	{attribute 'TcIecLibraryType'}
	{attribute 'external_name' := 'F_VN_GetAt_TcVnVector4_DINT_GUID_761AB84D_C513_5B06_61E4_80F931BBB792'}
	(* Gets the TcVnVector4_DINT element at the specified index of the container. *)
	FUNCTION F_VN_GetAt_TcVnVector4_DINT : HRESULT
	VAR_INPUT
		ipContainer	:	ITcVnContainer;	(* Container with TcVnVector4_DINT elements *)
		aElement	:	REFERENCE TO TcVnVector4_DINT;	(* Returns the element at the specified index *)
		nIndex	:	ULINT;	(* Index of the requested element *)
		hrPrev	:	HRESULT;	(* HRESULT indicating the result of previous operations (If SUCCEEDED(hrPrev) equals false, no operation is executed.) *)
	END_VAR

END_FUNCTION

// Functions/Basic Container Operations/F_VN_GetAt/F_VN_GetAt_TcVnVector4_LREAL

	{attribute 'TcIecLibraryType'}
	{attribute 'external_name' := 'F_VN_GetAt_TcVnVector4_LREAL_GUID_5FDC4290_5703_5BA7_61DD_065C1D8ADDFE'}
	(* Gets the TcVnVector4_LREAL element at the specified index of the container. *)
	FUNCTION F_VN_GetAt_TcVnVector4_LREAL : HRESULT
	VAR_INPUT
		ipContainer	:	ITcVnContainer;	(* Container with TcVnVector4_LREAL elements *)
		aElement	:	REFERENCE TO TcVnVector4_LREAL;	(* Returns the element at the specified index *)
		nIndex	:	ULINT;	(* Index of the requested element *)
		hrPrev	:	HRESULT;	(* HRESULT indicating the result of previous operations (If SUCCEEDED(hrPrev) equals false, no operation is executed.) *)
	END_VAR

END_FUNCTION

// Functions/Basic Container Operations/F_VN_GetAt/F_VN_GetAt_UDINT

	{attribute 'TcIecLibraryType'}
	{attribute 'external_name' := 'F_VN_GetAt_UDINT_GUID_C440DBA3_7390_5B33_575A_EBCC8FB96E53'}
	(* Gets the UDINT element at the specified index of the container. *)
	FUNCTION F_VN_GetAt_UDINT : HRESULT
	VAR_INPUT
		ipContainer	:	ITcVnContainer;	(* Container with UDINT elements *)
		nElement	:	REFERENCE TO UDINT;	(* Returns the element at the specified index *)
		nIndex	:	ULINT;	(* Index of the requested element *)
		hrPrev	:	HRESULT;	(* HRESULT indicating the result of previous operations (If SUCCEEDED(hrPrev) equals false, no operation is executed.) *)
	END_VAR

END_FUNCTION

// Functions/Basic Container Operations/F_VN_GetAt/F_VN_GetAt_ULINT

	{attribute 'TcIecLibraryType'}
	{attribute 'external_name' := 'F_VN_GetAt_ULINT_GUID_C7670D70_FA4B_5664_569F_3BAC6764E342'}
	(* Gets the ULINT element at the specified index of the container. *)
	FUNCTION F_VN_GetAt_ULINT : HRESULT
	VAR_INPUT
		ipContainer	:	ITcVnContainer;	(* Container with ULINT elements *)
		nElement	:	REFERENCE TO ULINT;	(* Returns the element at the specified index *)
		nIndex	:	ULINT;	(* Index of the requested element *)
		hrPrev	:	HRESULT;	(* HRESULT indicating the result of previous operations (If SUCCEEDED(hrPrev) equals false, no operation is executed.) *)
	END_VAR

END_FUNCTION

// Functions/Basic Container Operations/F_VN_InsertIntoContainer/F_VN_InsertIntoContainer_ITcVnContainer

	{attribute 'TcIecLibraryType'}
	{attribute 'external_name' := 'F_VN_InsertIntoContainer_ITcVnContainer_GUID_DDDC9785_B003_5B61_64D8_7B702B9B58A1'}
	(* Insert an element (or a range of elements) into a container before the specified position. *)
	FUNCTION F_VN_InsertIntoContainer_ITcVnContainer : HRESULT
	VAR_INPUT
		ipElement	:	ITcVnContainer;	(* Single element to insert into ipContainer or container with several elements *)
		ipContainer	:	ITcVnContainer;	(* Container in which to insert the element *)
		nIndex	:	ULINT;	(* Position, before which the element will be inserted *)
		hrPrev	:	HRESULT;	(* HRESULT indicating the result of previous operations (If SUCCEEDED(hrPrev) equals false, no operation is executed.) *)
	END_VAR

END_FUNCTION

// Functions/Basic Container Operations/F_VN_InsertIntoContainer/F_VN_InsertIntoContainer_ITcVnForwardIterator

	{attribute 'TcIecLibraryType'}
	{attribute 'external_name' := 'F_VN_InsertIntoContainer_ITcVnForwardIterator_GUID_80A27022_E316_5DC3_60F7_8E6960A418A2'}
	(* Insert an element (represented by an iterator) into a container before the specified position. *)
	FUNCTION F_VN_InsertIntoContainer_ITcVnForwardIterator : HRESULT
	VAR_INPUT
		ipElement	:	ITcVnForwardIterator;	(* Single element to insert into ipContainer *)
		ipContainer	:	ITcVnContainer;	(* Container in which to insert the element *)
		nIndex	:	ULINT;	(* Position, before which the element will be inserted *)
		hrPrev	:	HRESULT;	(* HRESULT indicating the result of previous operations (If SUCCEEDED(hrPrev) equals false, no operation is executed.) *)
	END_VAR

END_FUNCTION

// Functions/Basic Container Operations/F_VN_InsertIntoContainer/F_VN_InsertIntoContainer_DINT

	{attribute 'TcIecLibraryType'}
	{attribute 'external_name' := 'F_VN_InsertIntoContainer_DINT_GUID_EFA0F64D_773F_5851_76D4_98F1756231A4'}
	(* Insert an element of type DINT into a container before the specified position. *)
	FUNCTION F_VN_InsertIntoContainer_DINT : HRESULT
	VAR_INPUT
		nElement	:	DINT;	(* Single element to insert into ipContainer *)
		ipContainer	:	ITcVnContainer;	(* Container in which to insert the element *)
		nIndex	:	ULINT;	(* Position, before which the element will be inserted *)
		hrPrev	:	HRESULT;	(* HRESULT indicating the result of previous operations (If SUCCEEDED(hrPrev) equals false, no operation is executed.) *)
	END_VAR

END_FUNCTION

// Functions/Basic Container Operations/F_VN_InsertIntoContainer/F_VN_InsertIntoContainer_LREAL

	{attribute 'TcIecLibraryType'}
	{attribute 'external_name' := 'F_VN_InsertIntoContainer_LREAL_GUID_72B81CEB_6BEB_5915_6CF4_FBE0016B575A'}
	(* Insert an element of type LREAL into a container before the specified position. *)
	FUNCTION F_VN_InsertIntoContainer_LREAL : HRESULT
	VAR_INPUT
		fElement	:	LREAL;	(* Single element to insert into ipContainer *)
		ipContainer	:	ITcVnContainer;	(* Container in which to insert the element *)
		nIndex	:	ULINT;	(* Position, before which the element will be inserted *)
		hrPrev	:	HRESULT;	(* HRESULT indicating the result of previous operations (If SUCCEEDED(hrPrev) equals false, no operation is executed.) *)
	END_VAR

END_FUNCTION

// Functions/Basic Container Operations/F_VN_InsertIntoContainer/F_VN_InsertIntoContainer_REAL

	{attribute 'TcIecLibraryType'}
	{attribute 'external_name' := 'F_VN_InsertIntoContainer_REAL_GUID_3EA6CA06_995B_58CA_78EF_95938B01338C'}
	(* Insert an element of type REAL into a container before the specified position. *)
	FUNCTION F_VN_InsertIntoContainer_REAL : HRESULT
	VAR_INPUT
		fElement	:	REAL;	(* Single element to insert into ipContainer *)
		ipContainer	:	ITcVnContainer;	(* Container in which to insert the element *)
		nIndex	:	ULINT;	(* Position, before which the element will be inserted *)
		hrPrev	:	HRESULT;	(* HRESULT indicating the result of previous operations (If SUCCEEDED(hrPrev) equals false, no operation is executed.) *)
	END_VAR

END_FUNCTION

// Functions/Basic Container Operations/F_VN_InsertIntoContainer/F_VN_InsertIntoContainer_SINT

	{attribute 'TcIecLibraryType'}
	{attribute 'external_name' := 'F_VN_InsertIntoContainer_SINT_GUID_DC281E74_0A3E_5FA1_760C_538B9F283AFE'}
	(* Insert an element of type SINT into a container before the specified position. *)
	FUNCTION F_VN_InsertIntoContainer_SINT : HRESULT
	VAR_INPUT
		nElement	:	SINT;	(* Single element to insert into ipContainer *)
		ipContainer	:	ITcVnContainer;	(* Container in which to insert the element *)
		nIndex	:	ULINT;	(* Position, before which the element will be inserted *)
		hrPrev	:	HRESULT;	(* HRESULT indicating the result of previous operations (If SUCCEEDED(hrPrev) equals false, no operation is executed.) *)
	END_VAR

END_FUNCTION

// Functions/Basic Container Operations/F_VN_InsertIntoContainer/F_VN_InsertIntoContainer_TcVnDMatch

	{attribute 'TcIecLibraryType'}
	{attribute 'external_name' := 'F_VN_InsertIntoContainer_TcVnDMatch_GUID_6288EBFB_184C_50FA_5092_D3D94B3EFDC4'}
	(* Insert an element of type TcVnDMatch into a container before the specified position. *)
	FUNCTION F_VN_InsertIntoContainer_TcVnDMatch : HRESULT
	VAR_INPUT
		stElement	:	REFERENCE TO TcVnDMatch;	(* Single element to insert into ipContainer *)
		ipContainer	:	ITcVnContainer;	(* Container in which to insert the element *)
		nIndex	:	ULINT;	(* Position, before which the element will be inserted *)
		hrPrev	:	HRESULT;	(* HRESULT indicating the result of previous operations (If SUCCEEDED(hrPrev) equals false, no operation is executed.) *)
	END_VAR

END_FUNCTION

// Functions/Basic Container Operations/F_VN_InsertIntoContainer/F_VN_InsertIntoContainer_TcVnKeyPoint

	{attribute 'TcIecLibraryType'}
	{attribute 'external_name' := 'F_VN_InsertIntoContainer_TcVnKeyPoint_GUID_B6243C78_DA27_5D5E_5D78_25085B9D62AA'}
	(* Insert an element of type TcVnKeyPoint into a container before the specified position. *)
	FUNCTION F_VN_InsertIntoContainer_TcVnKeyPoint : HRESULT
	VAR_INPUT
		stElement	:	REFERENCE TO TcVnKeyPoint;	(* Single element to insert into ipContainer *)
		ipContainer	:	ITcVnContainer;	(* Container in which to insert the element *)
		nIndex	:	ULINT;	(* Position, before which the element will be inserted *)
		hrPrev	:	HRESULT;	(* HRESULT indicating the result of previous operations (If SUCCEEDED(hrPrev) equals false, no operation is executed.) *)
	END_VAR

END_FUNCTION

// Functions/Basic Container Operations/F_VN_InsertIntoContainer/F_VN_InsertIntoContainer_TcVnPoint2_DINT

	{attribute 'TcIecLibraryType'}
	{attribute 'external_name' := 'F_VN_InsertIntoContainer_TcVnPoint2_DINT_GUID_F549CEB7_E5A4_5BCF_494B_F1B410216754'}
	(* Insert an element of type TcVnPoint2_DINT into a container before the specified position. *)
	FUNCTION F_VN_InsertIntoContainer_TcVnPoint2_DINT : HRESULT
	VAR_INPUT
		aElement	:	REFERENCE TO TcVnPoint2_DINT;	(* Single element to insert into ipContainer *)
		ipContainer	:	ITcVnContainer;	(* Container in which to insert the element *)
		nIndex	:	ULINT;	(* Position, before which the element will be inserted *)
		hrPrev	:	HRESULT;	(* HRESULT indicating the result of previous operations (If SUCCEEDED(hrPrev) equals false, no operation is executed.) *)
	END_VAR

END_FUNCTION

// Functions/Basic Container Operations/F_VN_InsertIntoContainer/F_VN_InsertIntoContainer_TcVnPoint2_LREAL

	{attribute 'TcIecLibraryType'}
	{attribute 'external_name' := 'F_VN_InsertIntoContainer_TcVnPoint2_LREAL_GUID_0F32A540_CDF3_51E7_5F9A_C73CAA45BBE6'}
	(* Insert an element of type TcVnPoint2_LREAL into a container before the specified position. *)
	FUNCTION F_VN_InsertIntoContainer_TcVnPoint2_LREAL : HRESULT
	VAR_INPUT
		aElement	:	REFERENCE TO TcVnPoint2_LREAL;	(* Single element to insert into ipContainer *)
		ipContainer	:	ITcVnContainer;	(* Container in which to insert the element *)
		nIndex	:	ULINT;	(* Position, before which the element will be inserted *)
		hrPrev	:	HRESULT;	(* HRESULT indicating the result of previous operations (If SUCCEEDED(hrPrev) equals false, no operation is executed.) *)
	END_VAR

END_FUNCTION

// Functions/Basic Container Operations/F_VN_InsertIntoContainer/F_VN_InsertIntoContainer_TcVnPoint2_REAL

	{attribute 'TcIecLibraryType'}
	{attribute 'external_name' := 'F_VN_InsertIntoContainer_TcVnPoint2_REAL_GUID_727FB356_9228_5964_747E_75B2553FC054'}
	(* Insert an element of type TcVnPoint2_REAL into a container before the specified position. *)
	FUNCTION F_VN_InsertIntoContainer_TcVnPoint2_REAL : HRESULT
	VAR_INPUT
		aElement	:	REFERENCE TO TcVnPoint2_REAL;	(* Single element to insert into ipContainer *)
		ipContainer	:	ITcVnContainer;	(* Container in which to insert the element *)
		nIndex	:	ULINT;	(* Position, before which the element will be inserted *)
		hrPrev	:	HRESULT;	(* HRESULT indicating the result of previous operations (If SUCCEEDED(hrPrev) equals false, no operation is executed.) *)
	END_VAR

END_FUNCTION

// Functions/Basic Container Operations/F_VN_InsertIntoContainer/F_VN_InsertIntoContainer_TcVnPoint3_LREAL

	{attribute 'TcIecLibraryType'}
	{attribute 'external_name' := 'F_VN_InsertIntoContainer_TcVnPoint3_LREAL_GUID_0773769E_E9AF_5176_7931_BF10F0216404'}
	(* Insert an element of type TcVnPoint3_LREAL into a container before the specified position. *)
	FUNCTION F_VN_InsertIntoContainer_TcVnPoint3_LREAL : HRESULT
	VAR_INPUT
		aElement	:	REFERENCE TO TcVnPoint3_LREAL;	(* Single element to insert into ipContainer *)
		ipContainer	:	ITcVnContainer;	(* Container in which to insert the element *)
		nIndex	:	ULINT;	(* Position, before which the element will be inserted *)
		hrPrev	:	HRESULT;	(* HRESULT indicating the result of previous operations (If SUCCEEDED(hrPrev) equals false, no operation is executed.) *)
	END_VAR

END_FUNCTION

// Functions/Basic Container Operations/F_VN_InsertIntoContainer/F_VN_InsertIntoContainer_TcVnPoint3_REAL

	{attribute 'TcIecLibraryType'}
	{attribute 'external_name' := 'F_VN_InsertIntoContainer_TcVnPoint3_REAL_GUID_66633B0B_D08D_5FFD_5D37_7264CA3DA6E2'}
	(* Insert an element of type TcVnPoint3_REAL into a container before the specified position. *)
	FUNCTION F_VN_InsertIntoContainer_TcVnPoint3_REAL : HRESULT
	VAR_INPUT
		aElement	:	REFERENCE TO TcVnPoint3_REAL;	(* Single element to insert into ipContainer *)
		ipContainer	:	ITcVnContainer;	(* Container in which to insert the element *)
		nIndex	:	ULINT;	(* Position, before which the element will be inserted *)
		hrPrev	:	HRESULT;	(* HRESULT indicating the result of previous operations (If SUCCEEDED(hrPrev) equals false, no operation is executed.) *)
	END_VAR

END_FUNCTION

// Functions/Basic Container Operations/F_VN_InsertIntoContainer/F_VN_InsertIntoContainer_TcVnRectangle_DINT

	{attribute 'TcIecLibraryType'}
	{attribute 'external_name' := 'F_VN_InsertIntoContainer_TcVnRectangle_DINT_GUID_6D3C63D8_23BD_51A3_6598_36E39846907A'}
	(* Insert an element of type TcVnRectangle_DINT into a container before the specified position. *)
	FUNCTION F_VN_InsertIntoContainer_TcVnRectangle_DINT : HRESULT
	VAR_INPUT
		stElement	:	REFERENCE TO TcVnRectangle_DINT;	(* Single element to insert into ipContainer *)
		ipContainer	:	ITcVnContainer;	(* Container in which to insert the element *)
		nIndex	:	ULINT;	(* Position, before which the element will be inserted *)
		hrPrev	:	HRESULT;	(* HRESULT indicating the result of previous operations (If SUCCEEDED(hrPrev) equals false, no operation is executed.) *)
	END_VAR

END_FUNCTION

// Functions/Basic Container Operations/F_VN_InsertIntoContainer/F_VN_InsertIntoContainer_TcVnVector2_DINT

	{attribute 'TcIecLibraryType'}
	{attribute 'external_name' := 'F_VN_InsertIntoContainer_TcVnVector2_DINT_GUID_96D338D9_676E_50ED_60DB_FA4FFC7FDF34'}
	(* Insert an element of type TcVnVector2_DINT into a container before the specified position. *)
	FUNCTION F_VN_InsertIntoContainer_TcVnVector2_DINT : HRESULT
	VAR_INPUT
		aElement	:	REFERENCE TO TcVnVector2_DINT;	(* Single element to insert into ipContainer *)
		ipContainer	:	ITcVnContainer;	(* Container in which to insert the element *)
		nIndex	:	ULINT;	(* Position, before which the element will be inserted *)
		hrPrev	:	HRESULT;	(* HRESULT indicating the result of previous operations (If SUCCEEDED(hrPrev) equals false, no operation is executed.) *)
	END_VAR

END_FUNCTION

// Functions/Basic Container Operations/F_VN_InsertIntoContainer/F_VN_InsertIntoContainer_TcVnVector2_REAL

	{attribute 'TcIecLibraryType'}
	{attribute 'external_name' := 'F_VN_InsertIntoContainer_TcVnVector2_REAL_GUID_E74110AF_F945_5767_778B_24D2186D1C41'}
	(* Insert an element of type TcVnVector2_REAL into a container before the specified position. *)
	FUNCTION F_VN_InsertIntoContainer_TcVnVector2_REAL : HRESULT
	VAR_INPUT
		aElement	:	REFERENCE TO TcVnVector2_REAL;	(* Single element to insert into ipContainer *)
		ipContainer	:	ITcVnContainer;	(* Container in which to insert the element *)
		nIndex	:	ULINT;	(* Position, before which the element will be inserted *)
		hrPrev	:	HRESULT;	(* HRESULT indicating the result of previous operations (If SUCCEEDED(hrPrev) equals false, no operation is executed.) *)
	END_VAR

END_FUNCTION

// Functions/Basic Container Operations/F_VN_InsertIntoContainer/F_VN_InsertIntoContainer_TcVnVector3_REAL

	{attribute 'TcIecLibraryType'}
	{attribute 'external_name' := 'F_VN_InsertIntoContainer_TcVnVector3_REAL_GUID_7E113FC2_5BBC_54D7_6CFE_D698D46CE2A1'}
	(* Insert an element of type TcVnVector3_REAL into a container before the specified position. *)
	FUNCTION F_VN_InsertIntoContainer_TcVnVector3_REAL : HRESULT
	VAR_INPUT
		aElement	:	REFERENCE TO TcVnVector3_REAL;	(* Single element to insert into ipContainer *)
		ipContainer	:	ITcVnContainer;	(* Container in which to insert the element *)
		nIndex	:	ULINT;	(* Position, before which the element will be inserted *)
		hrPrev	:	HRESULT;	(* HRESULT indicating the result of previous operations (If SUCCEEDED(hrPrev) equals false, no operation is executed.) *)
	END_VAR

END_FUNCTION

// Functions/Basic Container Operations/F_VN_InsertIntoContainer/F_VN_InsertIntoContainer_TcVnVector4_DINT

	{attribute 'TcIecLibraryType'}
	{attribute 'external_name' := 'F_VN_InsertIntoContainer_TcVnVector4_DINT_GUID_4A3AD761_60B4_5081_5C01_BA7FAA99BCB9'}
	(* Insert an element of type TcVnVector4_DINT into a container before the specified position. *)
	FUNCTION F_VN_InsertIntoContainer_TcVnVector4_DINT : HRESULT
	VAR_INPUT
		aElement	:	REFERENCE TO TcVnVector4_DINT;	(* Single element to insert into ipContainer *)
		ipContainer	:	ITcVnContainer;	(* Container in which to insert the element *)
		nIndex	:	ULINT;	(* Position, before which the element will be inserted *)
		hrPrev	:	HRESULT;	(* HRESULT indicating the result of previous operations (If SUCCEEDED(hrPrev) equals false, no operation is executed.) *)
	END_VAR

END_FUNCTION

// Functions/Basic Container Operations/F_VN_InsertIntoContainer/F_VN_InsertIntoContainer_TcVnVector4_LREAL

	{attribute 'TcIecLibraryType'}
	{attribute 'external_name' := 'F_VN_InsertIntoContainer_TcVnVector4_LREAL_GUID_0DE3BAA5_BCB8_5749_62E9_D0780F00C723'}
	(* Insert an element of type TcVnVector4_LREAL into a container before the specified position. *)
	FUNCTION F_VN_InsertIntoContainer_TcVnVector4_LREAL : HRESULT
	VAR_INPUT
		aElement	:	REFERENCE TO TcVnVector4_LREAL;	(* Single element to insert into ipContainer *)
		ipContainer	:	ITcVnContainer;	(* Container in which to insert the element *)
		nIndex	:	ULINT;	(* Position, before which the element will be inserted *)
		hrPrev	:	HRESULT;	(* HRESULT indicating the result of previous operations (If SUCCEEDED(hrPrev) equals false, no operation is executed.) *)
	END_VAR

END_FUNCTION

// Functions/Basic Container Operations/F_VN_InsertIntoContainer/F_VN_InsertIntoContainer_UDINT

	{attribute 'TcIecLibraryType'}
	{attribute 'external_name' := 'F_VN_InsertIntoContainer_UDINT_GUID_B6D1E6FC_98F6_5CDB_5CC3_8811ED90DFDF'}
	(* Insert an element of type UDINT into a container before the specified position. *)
	FUNCTION F_VN_InsertIntoContainer_UDINT : HRESULT
	VAR_INPUT
		nElement	:	UDINT;	(* Single element to insert into ipContainer *)
		ipContainer	:	ITcVnContainer;	(* Container in which to insert the element *)
		nIndex	:	ULINT;	(* Position, before which the element will be inserted *)
		hrPrev	:	HRESULT;	(* HRESULT indicating the result of previous operations (If SUCCEEDED(hrPrev) equals false, no operation is executed.) *)
	END_VAR

END_FUNCTION

// Functions/Basic Container Operations/F_VN_InsertIntoContainer/F_VN_InsertIntoContainer_ULINT

	{attribute 'TcIecLibraryType'}
	{attribute 'external_name' := 'F_VN_InsertIntoContainer_ULINT_GUID_0DA88F93_3472_5D7A_5EDC_DFF2F9A1782F'}
	(* Insert an element of type ULINT into a container before the specified position. *)
	FUNCTION F_VN_InsertIntoContainer_ULINT : HRESULT
	VAR_INPUT
		nElement	:	ULINT;	(* Single element to insert into ipContainer *)
		ipContainer	:	ITcVnContainer;	(* Container in which to insert the element *)
		nIndex	:	ULINT;	(* Position, before which the element will be inserted *)
		hrPrev	:	HRESULT;	(* HRESULT indicating the result of previous operations (If SUCCEEDED(hrPrev) equals false, no operation is executed.) *)
	END_VAR

END_FUNCTION

// Functions/Basic Container Operations/F_VN_SetAt/F_VN_SetAt_ITcVnContainer

	{attribute 'TcIecLibraryType'}
	{attribute 'external_name' := 'F_VN_SetAt_ITcVnContainer_GUID_476292B8_B77C_54F1_6FFA_C3AAC9D44D9F'}
	(* Sets the element at the specified index of the container. (Alternatively use interface method .SetAt.) *)
	FUNCTION F_VN_SetAt_ITcVnContainer : HRESULT
	VAR_INPUT
		ipElement	:	ITcVnContainer;	(* Element to set at the specified container position *)
		ipContainer	:	ITcVnContainer;	(* Container with ITcVnContainer elements, in which the element at position nIndex is replaced by ipElement *)
		nIndex	:	ULINT;	(* Index *)
		hrPrev	:	HRESULT;	(* HRESULT indicating the result of previous operations (If SUCCEEDED(hrPrev) equals false, no operation is executed.) *)
	END_VAR

END_FUNCTION

// Functions/Basic Container Operations/F_VN_SetAt/F_VN_SetAt_DINT

	{attribute 'TcIecLibraryType'}
	{attribute 'external_name' := 'F_VN_SetAt_DINT_GUID_D681C79A_99FB_542C_5064_21278FC65E88'}
	(* Sets the element at the specified index of the container. *)
	FUNCTION F_VN_SetAt_DINT : HRESULT
	VAR_INPUT
		nElement	:	DINT;	(* Element to set at the specified container position *)
		ipContainer	:	ITcVnContainer;	(* Container with DINT elements, in which the element at position nIndex is replaced by nElement *)
		nIndex	:	ULINT;	(* Index *)
		hrPrev	:	HRESULT;	(* HRESULT indicating the result of previous operations (If SUCCEEDED(hrPrev) equals false, no operation is executed.) *)
	END_VAR

END_FUNCTION

// Functions/Basic Container Operations/F_VN_SetAt/F_VN_SetAt_LREAL

	{attribute 'TcIecLibraryType'}
	{attribute 'external_name' := 'F_VN_SetAt_LREAL_GUID_423656CE_3EEB_50CE_538A_C2294F8AC9E8'}
	(* Sets the element at the specified index of the container. *)
	FUNCTION F_VN_SetAt_LREAL : HRESULT
	VAR_INPUT
		fElement	:	LREAL;	(* Element to set at the specified container position *)
		ipContainer	:	ITcVnContainer;	(* Container with LREAL elements, in which the element at position nIndex is replaced by fElement *)
		nIndex	:	ULINT;	(* Index *)
		hrPrev	:	HRESULT;	(* HRESULT indicating the result of previous operations (If SUCCEEDED(hrPrev) equals false, no operation is executed.) *)
	END_VAR

END_FUNCTION

// Functions/Basic Container Operations/F_VN_SetAt/F_VN_SetAt_REAL

	{attribute 'TcIecLibraryType'}
	{attribute 'external_name' := 'F_VN_SetAt_REAL_GUID_8D20883B_2232_5CA0_46F3_1CAEEB220474'}
	(* Sets the element at the specified index of the container. *)
	FUNCTION F_VN_SetAt_REAL : HRESULT
	VAR_INPUT
		fElement	:	REAL;	(* Element to set at the specified container position *)
		ipContainer	:	ITcVnContainer;	(* Container with REAL elements, in which the element at position nIndex is replaced by fElement *)
		nIndex	:	ULINT;	(* Index *)
		hrPrev	:	HRESULT;	(* HRESULT indicating the result of previous operations (If SUCCEEDED(hrPrev) equals false, no operation is executed.) *)
	END_VAR

END_FUNCTION

// Functions/Basic Container Operations/F_VN_SetAt/F_VN_SetAt_SINT

	{attribute 'TcIecLibraryType'}
	{attribute 'external_name' := 'F_VN_SetAt_SINT_GUID_53FC7629_B651_5D0C_6E10_8210E70EB0CE'}
	(* Sets the element at the specified index of the container. *)
	FUNCTION F_VN_SetAt_SINT : HRESULT
	VAR_INPUT
		nElement	:	SINT;	(* Element to set at the specified container position *)
		ipContainer	:	ITcVnContainer;	(* Container with SINT elements, in which the element at position nIndex is replaced by nElement *)
		nIndex	:	ULINT;	(* Index *)
		hrPrev	:	HRESULT;	(* HRESULT indicating the result of previous operations (If SUCCEEDED(hrPrev) equals false, no operation is executed.) *)
	END_VAR

END_FUNCTION

// Functions/Basic Container Operations/F_VN_SetAt/F_VN_SetAt_TcVnDMatch

	{attribute 'TcIecLibraryType'}
	{attribute 'external_name' := 'F_VN_SetAt_TcVnDMatch_GUID_DE6374D9_34B5_5A1A_76F3_D708397AF9E9'}
	(* Sets the element at the specified index of the container. *)
	FUNCTION F_VN_SetAt_TcVnDMatch : HRESULT
	VAR_INPUT
		stElement	:	REFERENCE TO TcVnDMatch;	(* Element to set at the specified container position *)
		ipContainer	:	ITcVnContainer;	(* Container with TcVnDMatch elements, in which the element at position nIndex is replaced by stElement *)
		nIndex	:	ULINT;	(* Index *)
		hrPrev	:	HRESULT;	(* HRESULT indicating the result of previous operations (If SUCCEEDED(hrPrev) equals false, no operation is executed.) *)
	END_VAR

END_FUNCTION

// Functions/Basic Container Operations/F_VN_SetAt/F_VN_SetAt_TcVnKeyPoint

	{attribute 'TcIecLibraryType'}
	{attribute 'external_name' := 'F_VN_SetAt_TcVnKeyPoint_GUID_A6F74671_C5E7_5652_6D51_85B28D5B5475'}
	(* Sets the element at the specified index of the container. *)
	FUNCTION F_VN_SetAt_TcVnKeyPoint : HRESULT
	VAR_INPUT
		stElement	:	REFERENCE TO TcVnKeyPoint;	(* Element to set at the specified container position *)
		ipContainer	:	ITcVnContainer;	(* Container with TcVnKeyPoint elements, in which the element at position nIndex is replaced by stElement *)
		nIndex	:	ULINT;	(* Index *)
		hrPrev	:	HRESULT;	(* HRESULT indicating the result of previous operations (If SUCCEEDED(hrPrev) equals false, no operation is executed.) *)
	END_VAR

END_FUNCTION

// Functions/Basic Container Operations/F_VN_SetAt/F_VN_SetAt_TcVnPoint2_DINT

	{attribute 'TcIecLibraryType'}
	{attribute 'external_name' := 'F_VN_SetAt_TcVnPoint2_DINT_GUID_CBB9CE79_18E6_5A86_53EC_DCC9DA313DFD'}
	(* Sets the element at the specified index of the container. *)
	FUNCTION F_VN_SetAt_TcVnPoint2_DINT : HRESULT
	VAR_INPUT
		aElement	:	REFERENCE TO TcVnPoint2_DINT;	(* Element to set at the specified container position *)
		ipContainer	:	ITcVnContainer;	(* Container with TcVnPoint2_DINT elements, in which the element at position nIndex is replaced by aElement *)
		nIndex	:	ULINT;	(* Index *)
		hrPrev	:	HRESULT;	(* HRESULT indicating the result of previous operations (If SUCCEEDED(hrPrev) equals false, no operation is executed.) *)
	END_VAR

END_FUNCTION

// Functions/Basic Container Operations/F_VN_SetAt/F_VN_SetAt_TcVnPoint2_LREAL

	{attribute 'TcIecLibraryType'}
	{attribute 'external_name' := 'F_VN_SetAt_TcVnPoint2_LREAL_GUID_C0803B4C_5E0A_59E7_4B96_60DFDE71D332'}
	(* Sets the element at the specified index of the container. *)
	FUNCTION F_VN_SetAt_TcVnPoint2_LREAL : HRESULT
	VAR_INPUT
		aElement	:	REFERENCE TO TcVnPoint2_LREAL;	(* Element to set at the specified container position *)
		ipContainer	:	ITcVnContainer;	(* Container with TcVnPoint2_LREAL elements, in which the element at position nIndex is replaced by aElement *)
		nIndex	:	ULINT;	(* Index *)
		hrPrev	:	HRESULT;	(* HRESULT indicating the result of previous operations (If SUCCEEDED(hrPrev) equals false, no operation is executed.) *)
	END_VAR

END_FUNCTION

// Functions/Basic Container Operations/F_VN_SetAt/F_VN_SetAt_TcVnPoint2_REAL

	{attribute 'TcIecLibraryType'}
	{attribute 'external_name' := 'F_VN_SetAt_TcVnPoint2_REAL_GUID_9089A3D2_ECED_55A2_704E_02C6F5AC1EC2'}
	(* Sets the element at the specified index of the container. *)
	FUNCTION F_VN_SetAt_TcVnPoint2_REAL : HRESULT
	VAR_INPUT
		aElement	:	REFERENCE TO TcVnPoint2_REAL;	(* Element to set at the specified container position *)
		ipContainer	:	ITcVnContainer;	(* Container with TcVnPoint2_REAL elements, in which the element at position nIndex is replaced by aElement *)
		nIndex	:	ULINT;	(* Index *)
		hrPrev	:	HRESULT;	(* HRESULT indicating the result of previous operations (If SUCCEEDED(hrPrev) equals false, no operation is executed.) *)
	END_VAR

END_FUNCTION

// Functions/Basic Container Operations/F_VN_SetAt/F_VN_SetAt_TcVnPoint3_LREAL

	{attribute 'TcIecLibraryType'}
	{attribute 'external_name' := 'F_VN_SetAt_TcVnPoint3_LREAL_GUID_09B386C3_A97A_58B8_78DB_33FA210F652E'}
	(* Sets the element at the specified index of the container. *)
	FUNCTION F_VN_SetAt_TcVnPoint3_LREAL : HRESULT
	VAR_INPUT
		aElement	:	REFERENCE TO TcVnPoint3_LREAL;	(* Element to set at the specified container position *)
		ipContainer	:	ITcVnContainer;	(* Container with TcVnPoint3_LREAL elements, in which the element at position nIndex is replaced by aElement *)
		nIndex	:	ULINT;	(* Index *)
		hrPrev	:	HRESULT;	(* HRESULT indicating the result of previous operations (If SUCCEEDED(hrPrev) equals false, no operation is executed.) *)
	END_VAR

END_FUNCTION

// Functions/Basic Container Operations/F_VN_SetAt/F_VN_SetAt_TcVnPoint3_REAL

	{attribute 'TcIecLibraryType'}
	{attribute 'external_name' := 'F_VN_SetAt_TcVnPoint3_REAL_GUID_3AA6ED5C_D431_57BB_42D3_FC455BD67AEE'}
	(* Sets the element at the specified index of the container. *)
	FUNCTION F_VN_SetAt_TcVnPoint3_REAL : HRESULT
	VAR_INPUT
		aElement	:	REFERENCE TO TcVnPoint3_REAL;	(* Element to set at the specified container position *)
		ipContainer	:	ITcVnContainer;	(* Container with TcVnPoint3_REAL elements, in which the element at position nIndex is replaced by aElement *)
		nIndex	:	ULINT;	(* Index *)
		hrPrev	:	HRESULT;	(* HRESULT indicating the result of previous operations (If SUCCEEDED(hrPrev) equals false, no operation is executed.) *)
	END_VAR

END_FUNCTION

// Functions/Basic Container Operations/F_VN_SetAt/F_VN_SetAt_TcVnRectangle_DINT

	{attribute 'TcIecLibraryType'}
	{attribute 'external_name' := 'F_VN_SetAt_TcVnRectangle_DINT_GUID_B6875C80_57A2_53FA_62B0_D1707619700F'}
	(* Sets the element at the specified index of the container. *)
	FUNCTION F_VN_SetAt_TcVnRectangle_DINT : HRESULT
	VAR_INPUT
		stElement	:	REFERENCE TO TcVnRectangle_DINT;	(* Element to set at the specified container position *)
		ipContainer	:	ITcVnContainer;	(* Container with TcVnRectangle_DINT elements, in which the element at position nIndex is replaced by stElement *)
		nIndex	:	ULINT;	(* Index *)
		hrPrev	:	HRESULT;	(* HRESULT indicating the result of previous operations (If SUCCEEDED(hrPrev) equals false, no operation is executed.) *)
	END_VAR

END_FUNCTION

// Functions/Basic Container Operations/F_VN_SetAt/F_VN_SetAt_TcVnVector2_DINT

	{attribute 'TcIecLibraryType'}
	{attribute 'external_name' := 'F_VN_SetAt_TcVnVector2_DINT_GUID_DD29B9CC_1FA7_59DE_5D6A_4BD213537E38'}
	(* Sets the element at the specified index of the container. *)
	FUNCTION F_VN_SetAt_TcVnVector2_DINT : HRESULT
	VAR_INPUT
		aElement	:	REFERENCE TO TcVnVector2_DINT;	(* Element to set at the specified container position *)
		ipContainer	:	ITcVnContainer;	(* Container with TcVnVector2_DINT elements, in which the element at position nIndex is replaced by aElement *)
		nIndex	:	ULINT;	(* Index *)
		hrPrev	:	HRESULT;	(* HRESULT indicating the result of previous operations (If SUCCEEDED(hrPrev) equals false, no operation is executed.) *)
	END_VAR

END_FUNCTION

// Functions/Basic Container Operations/F_VN_SetAt/F_VN_SetAt_TcVnVector2_REAL

	{attribute 'TcIecLibraryType'}
	{attribute 'external_name' := 'F_VN_SetAt_TcVnVector2_REAL_GUID_0F5B0DA0_1480_5F68_5940_945F4CF7A15F'}
	(* Sets the element at the specified index of the container. *)
	FUNCTION F_VN_SetAt_TcVnVector2_REAL : HRESULT
	VAR_INPUT
		aElement	:	REFERENCE TO TcVnVector2_REAL;	(* Element to set at the specified container position *)
		ipContainer	:	ITcVnContainer;	(* Container with TcVnVector2_REAL elements, in which the element at position nIndex is replaced by aElement *)
		nIndex	:	ULINT;	(* Index *)
		hrPrev	:	HRESULT;	(* HRESULT indicating the result of previous operations (If SUCCEEDED(hrPrev) equals false, no operation is executed.) *)
	END_VAR

END_FUNCTION

// Functions/Basic Container Operations/F_VN_SetAt/F_VN_SetAt_TcVnVector3_REAL

	{attribute 'TcIecLibraryType'}
	{attribute 'external_name' := 'F_VN_SetAt_TcVnVector3_REAL_GUID_1454F9B4_0602_5B69_5941_414084146024'}
	(* Sets the element at the specified index of the container. *)
	FUNCTION F_VN_SetAt_TcVnVector3_REAL : HRESULT
	VAR_INPUT
		aElement	:	REFERENCE TO TcVnVector3_REAL;	(* Element to set at the specified container position *)
		ipContainer	:	ITcVnContainer;	(* Container with TcVnVector3_REAL elements, in which the element at position nIndex is replaced by aElement *)
		nIndex	:	ULINT;	(* Index *)
		hrPrev	:	HRESULT;	(* HRESULT indicating the result of previous operations (If SUCCEEDED(hrPrev) equals false, no operation is executed.) *)
	END_VAR

END_FUNCTION

// Functions/Basic Container Operations/F_VN_SetAt/F_VN_SetAt_TcVnVector4_DINT

	{attribute 'TcIecLibraryType'}
	{attribute 'external_name' := 'F_VN_SetAt_TcVnVector4_DINT_GUID_072C4DDC_9BFD_5FA3_4604_24EC0CFA6015'}
	(* Sets the element at the specified index of the container. *)
	FUNCTION F_VN_SetAt_TcVnVector4_DINT : HRESULT
	VAR_INPUT
		aElement	:	REFERENCE TO TcVnVector4_DINT;	(* Element to set at the specified container position *)
		ipContainer	:	ITcVnContainer;	(* Container with TcVnVector4_DINT elements, in which the element at position nIndex is replaced by aElement *)
		nIndex	:	ULINT;	(* Index *)
		hrPrev	:	HRESULT;	(* HRESULT indicating the result of previous operations (If SUCCEEDED(hrPrev) equals false, no operation is executed.) *)
	END_VAR

END_FUNCTION

// Functions/Basic Container Operations/F_VN_SetAt/F_VN_SetAt_TcVnVector4_LREAL

	{attribute 'TcIecLibraryType'}
	{attribute 'external_name' := 'F_VN_SetAt_TcVnVector4_LREAL_GUID_30AA56D9_7C3C_5666_4E1F_B45235D14E59'}
	(* Sets the element at the specified index of the container. *)
	FUNCTION F_VN_SetAt_TcVnVector4_LREAL : HRESULT
	VAR_INPUT
		aElement	:	REFERENCE TO TcVnVector4_LREAL;	(* Element to set at the specified container position *)
		ipContainer	:	ITcVnContainer;	(* Container with TcVnVector4_LREAL elements, in which the element at position nIndex is replaced by aElement *)
		nIndex	:	ULINT;	(* Index *)
		hrPrev	:	HRESULT;	(* HRESULT indicating the result of previous operations (If SUCCEEDED(hrPrev) equals false, no operation is executed.) *)
	END_VAR

END_FUNCTION

// Functions/Basic Container Operations/F_VN_SetAt/F_VN_SetAt_UDINT

	{attribute 'TcIecLibraryType'}
	{attribute 'external_name' := 'F_VN_SetAt_UDINT_GUID_40B05280_973C_5DCE_4051_62D4C4E38F07'}
	(* Sets the element at the specified index of the container. *)
	FUNCTION F_VN_SetAt_UDINT : HRESULT
	VAR_INPUT
		nElement	:	UDINT;	(* Element to set at the specified container position *)
		ipContainer	:	ITcVnContainer;	(* Container with UDINT elements, in which the element at position nIndex is replaced by nElement *)
		nIndex	:	ULINT;	(* Index *)
		hrPrev	:	HRESULT;	(* HRESULT indicating the result of previous operations (If SUCCEEDED(hrPrev) equals false, no operation is executed.) *)
	END_VAR

END_FUNCTION

// Functions/Basic Container Operations/F_VN_SetAt/F_VN_SetAt_ULINT

	{attribute 'TcIecLibraryType'}
	{attribute 'external_name' := 'F_VN_SetAt_ULINT_GUID_7FA306F3_87E6_5EB8_7DF2_7DE9EA11E389'}
	(* Sets the element at the specified index of the container. *)
	FUNCTION F_VN_SetAt_ULINT : HRESULT
	VAR_INPUT
		nElement	:	ULINT;	(* Element to set at the specified container position *)
		ipContainer	:	ITcVnContainer;	(* Container with ULINT elements, in which the element at position nIndex is replaced by nElement *)
		nIndex	:	ULINT;	(* Index *)
		hrPrev	:	HRESULT;	(* HRESULT indicating the result of previous operations (If SUCCEEDED(hrPrev) equals false, no operation is executed.) *)
	END_VAR

END_FUNCTION

// Functions/Geometric and Coordinate Transformations/Calibration/F_VN_CalibrateCamera

	{attribute 'TcIecLibraryType'}
	{attribute 'external_name' := 'F_VN_CalibrateCamera_GUID_689A4FD0_3F8C_52A9_6DE2_058A6325749E'}
	(* Compute the camera parameters (intrinsic + extrinsic) by evaluating an image containing a calibration pattern (circles). *)
	FUNCTION F_VN_CalibrateCamera : HRESULT
	VAR_INPUT
		ipSrcImage	:	ITcVnImage;	(* Source image containing a calibration pattern (1 channel, USINT elements) *)
		ipReferencePoints	:	ITcVnContainer;	(* Reference calibration pattern point positions (ContainerType_Vector_TcVnPoint3_REAL) *)
		aCameraMatrix	:	REFERENCE TO TcVnMatrix3x3_LREAL;	(* Returns the camera matrix *)
		aDistortionCoefficients	:	REFERENCE TO TcVnArray8_LREAL;	(* Returns the lens distortion coefficients [k1, k2, p1, p2, k3, k4, k5, k6] *)
		aRotationMatrix	:	REFERENCE TO TcVnMatrix3x3_LREAL;	(* Returns the rotation matrix *)
		aTranslationVector	:	REFERENCE TO TcVnVector3_LREAL;	(* Returns the translation vector *)
		fReprojError	:	REFERENCE TO LREAL;	(* Returns the reprojection error *)
		stBlobDetectionParams	:	REFERENCE TO TcVnParamsBlobDetection;	(* Parameters for the internally used F_VN_DetectBlobs function *)
		stCalibrationOptions	:	REFERENCE TO TcVnCameraCalibrationOptions;	(* Calibration options *)
		hrPrev	:	HRESULT;	(* HRESULT indicating the result of previous operations (If SUCCEEDED(hrPrev) equals false, no operation is executed.) *)
	END_VAR

END_FUNCTION

// Functions/Geometric and Coordinate Transformations/Calibration/F_VN_CalibrateCameraExp

	{attribute 'TcIecLibraryType'}
	{attribute 'external_name' := 'F_VN_CalibrateCameraExp_GUID_9E4F8F39_C817_5DF3_763A_2115BCB02FB8'}
	(* Compute the camera parameters (intrinsic + extrinsic) by evaluating images containing a calibration pattern (circles). The extrinsic parameters are computed for the first image in the array. (expert function) *)
	FUNCTION F_VN_CalibrateCameraExp : HRESULT
	VAR_INPUT
		pSrcImages	:	PVOID;	(* Pointer to an array of source images, each containing the same calibration pattern (1 channel, USINT elements) *)
		nSrcArraySize	:	UINT;	(* pSrcImages array size *)
		ipReferencePoints	:	ITcVnContainer;	(* Reference calibration pattern point positions (ContainerType_Vector_TcVnPoint3_REAL) *)
		aCameraMatrix	:	REFERENCE TO TcVnMatrix3x3_LREAL;	(* Returns the camera matrix *)
		aDistortionCoefficients	:	REFERENCE TO TcVnArray8_LREAL;	(* Returns the lens distortion coefficients [k1, k2, p1, p2, k3, k4, k5, k6] *)
		aRotationMatrix	:	REFERENCE TO TcVnMatrix3x3_LREAL;	(* Returns the rotation matrix *)
		aTranslationVector	:	REFERENCE TO TcVnVector3_LREAL;	(* Returns the translation vector *)
		fReprojError	:	REFERENCE TO LREAL;	(* Returns the reprojection error *)
		stBlobDetectionParams	:	REFERENCE TO TcVnParamsBlobDetection;	(* Parameters for the internally used F_VN_DetectBlobs function *)
		stCalibrationOptions	:	REFERENCE TO TcVnCameraCalibrationOptions;	(* Calibration options *)
		hrPrev	:	HRESULT;	(* HRESULT indicating the result of previous operations (If SUCCEEDED(hrPrev) equals false, no operation is executed.) *)
	END_VAR

END_FUNCTION

// Functions/Geometric and Coordinate Transformations/Calibration/F_VN_CalibrateCameraManually

	{attribute 'TcIecLibraryType'}
	{attribute 'external_name' := 'F_VN_CalibrateCameraManually_GUID_DE881DBF_7F98_560E_6A5A_763C7B294004'}
	(* Compute the camera parameters (intrinsic + extrinsic). *)
	FUNCTION F_VN_CalibrateCameraManually : HRESULT
	VAR_INPUT
		ipImagePoints	:	ITcVnContainer;	(* Provided image points of multiple images (ContainerType_Vector_Vector_TcVnPoint2_REAL, each inner container with at least 4 points, same order as in ipReferencePoints) *)
		nImageWidth	:	UDINT;	(* Image width *)
		nImageHeight	:	UDINT;	(* Image height *)
		ipReferencePoints	:	ITcVnContainer;	(* Reference world points (ContainerType_Vector_Vector_TcVnPoint3_REAL, same amount of points as ipImagePoints) *)
		aCameraMatrix	:	REFERENCE TO TcVnMatrix3x3_LREAL;	(* Returns the camera matrix *)
		aDistortionCoefficients	:	REFERENCE TO TcVnArray8_LREAL;	(* Returns the lens distortion coefficients [k1, k2, p1, p2, k3, k4, k5, k6] *)
		aRotationMatrix	:	REFERENCE TO TcVnMatrix3x3_LREAL;	(* Returns the rotation matrix *)
		aTranslationVector	:	REFERENCE TO TcVnVector3_LREAL;	(* Returns the translation vector *)
		fReprojError	:	REFERENCE TO LREAL;	(* Returns the reprojection error *)
		stCalibrationOptions	:	REFERENCE TO TcVnCameraCalibrationOptions;	(* Calibration options *)
		hrPrev	:	HRESULT;	(* HRESULT indicating the result of previous operations (If SUCCEEDED(hrPrev) equals false, no operation is executed.) *)
	END_VAR

END_FUNCTION

// Functions/Geometric and Coordinate Transformations/Calibration/F_VN_CalibrateCameraPlanar

	{attribute 'TcIecLibraryType'}
	{attribute 'external_name' := 'F_VN_CalibrateCameraPlanar_GUID_5EA61155_E866_5827_428A_3D35396EE97C'}
	(* Calibrate camera using a planar calibration pattern comprised of four circles marking the corners of a rectangle. *)
	FUNCTION F_VN_CalibrateCameraPlanar : HRESULT
	VAR_INPUT
		ipSrcImage	:	ITcVnImage;	(* Binary source image (background zero, markers non-zero) *)
		aMarkerPositions	:	REFERENCE TO TcVnArray4_Point2_REAL;	(* Marker positions within their plane using world units (right-handed coordinate system) *)
		aTransformationMatrix	:	REFERENCE TO TcVnMatrix3x3_LREAL;	(* Returns a 3-by-3 matrix for the transformation from image coordinates into the reference coordinate system *)
		hrPrev	:	HRESULT;	(* HRESULT indicating the result of previous operations (If SUCCEEDED(hrPrev) equals false, no operation is executed.) *)
	END_VAR

END_FUNCTION

// Functions/Geometric and Coordinate Transformations/Calibration/F_VN_CalibrateCameraPlanarExp

	{attribute 'TcIecLibraryType'}
	{attribute 'external_name' := 'F_VN_CalibrateCameraPlanarExp_GUID_FEC1C597_273C_5520_575C_D0D2115421C4'}
	(* Calibrate camera using a planar calibration pattern comprised of four circles marking the corners of a rectangle. (expert function) *)
	FUNCTION F_VN_CalibrateCameraPlanarExp : HRESULT
	VAR_INPUT
		ipSrcImage	:	ITcVnImage;	(* Binary source image (background zero, markers non-zero) *)
		aMarkerPositions	:	REFERENCE TO TcVnArray4_Point2_REAL;	(* Marker positions within their plane using world units (right-handed coordinate system) *)
		aTransformationMatrix	:	REFERENCE TO TcVnMatrix3x3_LREAL;	(* Returns a 3-by-3 matrix for the transformation from image coordinates into the reference coordinate system *)
		aMarkerImagePositions	:	REFERENCE TO TcVnArray4_Point2_REAL;	(* Returns the marker positions in image coordinates (left-handed coordinate system) *)
		nMinMarkerArea	:	UDINT;	(* Minimum area for the detection of markers (Smaller markers are ignored.) *)
		nMaxMarkerArea	:	UDINT;	(* Maximum area for the detection of markers (Larger markers are ignored.) *)
		fMaxMarkerEccentricity	:	LREAL;	(* Maximum eccenticity for the detection of markers (The eccentricity measures deviations from a round shape (eccentricity = 0: round object; eccentricity = 1.0:  linear object).) *)
		hrPrev	:	HRESULT;	(* HRESULT indicating the result of previous operations (If SUCCEEDED(hrPrev) equals false, no operation is executed.) *)
	END_VAR

END_FUNCTION

// Functions/Geometric and Coordinate Transformations/Calibration/F_VN_CompensateLensDistortion

	{attribute 'TcIecLibraryType'}
	{attribute 'external_name' := 'F_VN_CompensateLensDistortion_GUID_CBB1E0C9_72E1_5B3E_7EB2_FD89B201A4A5'}
	(* Transforms an image to compensate the lens distortion. *)
	FUNCTION F_VN_CompensateLensDistortion : HRESULT
	VAR_INPUT
		ipSrcImage	:	ITcVnImage;	(* Source image *)
		ipDestImage	:	REFERENCE TO ITcVnImage;	(* Destination image (An appropriate destination image will be created if required.) *)
		aCameraMatrix	:	REFERENCE TO TcVnMatrix3x3_LREAL;	(* Camera matrix containing the intrinsic parameters *)
		aDistortionCoefficients	:	REFERENCE TO TcVnArray4_LREAL;	(* Lens distortion coefficients [k1, k2, p1, p2] *)
		hrPrev	:	HRESULT;	(* HRESULT indicating the result of previous operations (If SUCCEEDED(hrPrev) equals false, no operation is executed.) *)
	END_VAR

END_FUNCTION

// Functions/Geometric and Coordinate Transformations/Calibration/F_VN_CompensateLensDistortionExp1

	{attribute 'TcIecLibraryType'}
	{attribute 'external_name' := 'F_VN_CompensateLensDistortionExp1_GUID_51CC86CE_2EC2_5725_7926_EA4CF3599825'}
	(* Transforms an image to compensate the lens distortion. (expert function) *)
	FUNCTION F_VN_CompensateLensDistortionExp1 : HRESULT
	VAR_INPUT
		ipSrcImage	:	ITcVnImage;	(* Source image *)
		ipDestImage	:	REFERENCE TO ITcVnImage;	(* Destination image (An appropriate destination image will be created if required.) *)
		aCameraMatrix	:	REFERENCE TO TcVnMatrix3x3_LREAL;	(* Camera matrix containing the intrinsic parameters *)
		aDistortionCoefficients	:	REFERENCE TO TcVnArray8_LREAL;	(* Lens distortion coefficients [k1, k2, p1, p2, k3, k4, k5, k6] *)
		hrPrev	:	HRESULT;	(* HRESULT indicating the result of previous operations (If SUCCEEDED(hrPrev) equals false, no operation is executed.) *)
	END_VAR

END_FUNCTION

// Functions/Geometric and Coordinate Transformations/Calibration/F_VN_CompensateLensDistortionExp2

	{attribute 'TcIecLibraryType'}
	{attribute 'external_name' := 'F_VN_CompensateLensDistortionExp2_GUID_AE57D942_6BC7_5727_5D22_454B8EF06455'}
	(* Transforms an image to compensate the lens distortion. (expert function) *)
	FUNCTION F_VN_CompensateLensDistortionExp2 : HRESULT
	VAR_INPUT
		ipSrcImage	:	ITcVnImage;	(* Source image *)
		ipDestImage	:	REFERENCE TO ITcVnImage;	(* Destination image (An appropriate destination image will be created if required.) *)
		aCameraMatrix	:	REFERENCE TO TcVnMatrix3x3_LREAL;	(* Camera matrix containing the intrinsic parameters *)
		aDistortionCoefficients	:	REFERENCE TO TcVnArray8_LREAL;	(* Lens distortion coefficients [k1, k2, p1, p2, k3, k4, k5, k6] *)
		aNewCameraMatrix	:	REFERENCE TO TcVnMatrix3x3_LREAL;	(* Allows additional scaling and shifting of the result image *)
		hrPrev	:	HRESULT;	(* HRESULT indicating the result of previous operations (If SUCCEEDED(hrPrev) equals false, no operation is executed.) *)
	END_VAR

END_FUNCTION

// Functions/Geometric and Coordinate Transformations/Calibration/F_VN_CompensateLensDistortionForPoints

	{attribute 'TcIecLibraryType'}
	{attribute 'external_name' := 'F_VN_CompensateLensDistortionForPoints_GUID_76295BA5_956B_5713_4503_6A5E53895B3F'}
	(* Transforms point coordinates to compensate the lens distortion. *)
	FUNCTION F_VN_CompensateLensDistortionForPoints : HRESULT
	VAR_INPUT
		ipSrcPoints	:	ITcVnContainer;	(* Container with source point coordinates (ContainerType_Vector_TcVnPoint2_REAL or ContainerType_Vector_TcVnPoint2_DINT) *)
		ipDestPoints	:	REFERENCE TO ITcVnContainer;	(* Returns a container with the transformed point coordinates (ContainerType_Vector_TcVnPoint2_REAL) *)
		aCameraMatrix	:	REFERENCE TO TcVnMatrix3x3_LREAL;	(* Camera matrix containing the intrinsic parameters *)
		aDistortionCoefficients	:	REFERENCE TO TcVnArray4_LREAL;	(* Lens distortion coefficients [k1, k2, p1, p2] *)
		hrPrev	:	HRESULT;	(* HRESULT indicating the result of previous operations (If SUCCEEDED(hrPrev) equals false, no operation is executed.) *)
	END_VAR

END_FUNCTION

// Functions/Geometric and Coordinate Transformations/Calibration/F_VN_CompensateLensDistortionForPointsExp1

	{attribute 'TcIecLibraryType'}
	{attribute 'external_name' := 'F_VN_CompensateLensDistortionForPointsExp1_GUID_17DC8C11_965C_573B_7421_45C78A98F0B1'}
	(* Transforms point coordinates to compensate the lens distortion. (expert function) *)
	FUNCTION F_VN_CompensateLensDistortionForPointsExp1 : HRESULT
	VAR_INPUT
		ipSrcPoints	:	ITcVnContainer;	(* Container with source point coordinates (ContainerType_Vector_TcVnPoint2_REAL or ContainerType_Vector_TcVnPoint2_DINT) *)
		ipDestPoints	:	REFERENCE TO ITcVnContainer;	(* Returns a container with the transformed point coordinates (ContainerType_Vector_TcVnPoint2_REAL) *)
		aCameraMatrix	:	REFERENCE TO TcVnMatrix3x3_LREAL;	(* Camera matrix containing the intrinsic parameters *)
		aDistortionCoefficients	:	REFERENCE TO TcVnArray8_LREAL;	(* Lens distortion coefficients [k1, k2, p1, p2, k3, k4, k5, k6] *)
		hrPrev	:	HRESULT;	(* HRESULT indicating the result of previous operations (If SUCCEEDED(hrPrev) equals false, no operation is executed.) *)
	END_VAR

END_FUNCTION

// Functions/Geometric and Coordinate Transformations/Calibration/F_VN_CompensateLensDistortionForPointsExp2

	{attribute 'TcIecLibraryType'}
	{attribute 'external_name' := 'F_VN_CompensateLensDistortionForPointsExp2_GUID_580DD8FE_232B_5D0F_56A5_CB616AB70164'}
	(* Transforms point coordinates to compensate the lens distortion. (expert function) *)
	FUNCTION F_VN_CompensateLensDistortionForPointsExp2 : HRESULT
	VAR_INPUT
		ipSrcPoints	:	ITcVnContainer;	(* Container with source point coordinates (ContainerType_Vector_TcVnPoint2_REAL or ContainerType_Vector_TcVnPoint2_DINT) *)
		ipDestPoints	:	REFERENCE TO ITcVnContainer;	(* Returns a container with the transformed point coordinates (ContainerType_Vector_TcVnPoint2_REAL) *)
		aCameraMatrix	:	REFERENCE TO TcVnMatrix3x3_LREAL;	(* Camera matrix containing the intrinsic parameters *)
		aDistortionCoefficients	:	REFERENCE TO TcVnArray8_LREAL;	(* Lens distortion coefficients [k1, k2, p1, p2, k3, k4, k5, k6] *)
		aNewCameraMatrix	:	REFERENCE TO TcVnMatrix3x3_LREAL;	(* Allows additional shifting of the result point coordinates *)
		hrPrev	:	HRESULT;	(* HRESULT indicating the result of previous operations (If SUCCEEDED(hrPrev) equals false, no operation is executed.) *)
	END_VAR

END_FUNCTION

// Functions/Geometric and Coordinate Transformations/Calibration/F_VN_TransformCoordinatesPlanar_Container

	{attribute 'TcIecLibraryType'}
	{attribute 'external_name' := 'F_VN_TransformCoordinatesPlanar_Container_GUID_0B0CC95B_F42B_5C42_6508_29E6B8063DF0'}
	(* Compute real-world coordinates for given image points or vice versa. *)
	FUNCTION F_VN_TransformCoordinatesPlanar_Container : HRESULT
	VAR_INPUT
		ipSrcPoints	:	ITcVnContainer;	(* Container with 2D source points (TcVnPoint2_DINT or TcVnPoint2_REAL or TcVnPoint2_LREAL) *)
		ipDestPoints	:	REFERENCE TO ITcVnContainer;	(* Returns the transformed 2D points (TcVnPoint2_LREAL) *)
		aTransformationMatrix	:	REFERENCE TO TcVnMatrix3x3_LREAL;	(* Transformation matrix obtained with VnCalibrateCameraPlanar() or its inverse matrix obtained with VnInvertMatrix3x3() *)
		hrPrev	:	HRESULT;	(* HRESULT indicating the result of previous operations (If SUCCEEDED(hrPrev) equals false, no operation is executed.) *)
	END_VAR

END_FUNCTION

// Functions/Geometric and Coordinate Transformations/Calibration/F_VN_TransformCoordinatesPlanar_Point

	{attribute 'TcIecLibraryType'}
	{attribute 'external_name' := 'F_VN_TransformCoordinatesPlanar_Point_GUID_FFF67447_DBD8_5FA8_6BD4_F8748C59BC0A'}
	(* Compute real-world coordinates for a given image point or vice versa. *)
	FUNCTION F_VN_TransformCoordinatesPlanar_Point : HRESULT
	VAR_INPUT
		aSrcPoint	:	REFERENCE TO TcVnPoint2_LREAL;	(* Point in the source coordinate system *)
		aDestPoint	:	REFERENCE TO TcVnPoint2_LREAL;	(* Returns point in the destination coordinate system *)
		aTransformationMatrix	:	REFERENCE TO TcVnMatrix3x3_LREAL;	(* Transformation matrix obtained with VnCalibrateCameraPlanar() or its inverse matrix obtained with VnInvertMatrix3x3() *)
		hrPrev	:	HRESULT;	(* HRESULT indicating the result of previous operations (If SUCCEEDED(hrPrev) equals false, no operation is executed.) *)
	END_VAR

END_FUNCTION

// Functions/Geometric and Coordinate Transformations/Calibration/F_VN_TransformCoordinatesImageToWorld_Container

	{attribute 'TcIecLibraryType'}
	{attribute 'external_name' := 'F_VN_TransformCoordinatesImageToWorld_Container_GUID_389B6CAE_805D_5DE7_5A22_E1B341FFCFBA'}
	(* Transform 2D image point coordinates to 3D world coordinates (using intrinsic + extrinsic calibration results). *)
	FUNCTION F_VN_TransformCoordinatesImageToWorld_Container : HRESULT
	VAR_INPUT
		ipSrcPoints2D	:	ITcVnContainer;	(* Container with 2D source points (TcVnPoint2_DINT or TcVnPoint2_REAL or TcVnPoint2_LREAL) *)
		ipDestPoints3D	:	REFERENCE TO ITcVnContainer;	(* Returns the transformed 3D points (TcVnPoint3_LREAL) *)
		aCameraMatrix	:	REFERENCE TO TcVnMatrix3x3_LREAL;	(* 3x3 camera matrix containing the intrinsic parameters *)
		aDistortionCoefficients	:	REFERENCE TO TcVnArray8_LREAL;	(* Lens distortion coefficients [k1, k2, p1, p2, k3, k4, k5, k6] *)
		aRotationMatrix	:	REFERENCE TO TcVnMatrix3x3_LREAL;	(* 3x3 rotation matrix *)
		aTranslationVector	:	REFERENCE TO TcVnVector3_LREAL;	(* Translation vector *)
		fZ	:	LREAL;	(* z coordinate (world coordinate system) of the transformed points (0 would be at (toplevel) calibration pattern) *)
		hrPrev	:	HRESULT;	(* HRESULT indicating the result of previous operations (If SUCCEEDED(hrPrev) equals false, no operation is executed.) *)
	END_VAR

END_FUNCTION

// Functions/Geometric and Coordinate Transformations/Calibration/F_VN_TransformCoordinatesImageToWorld_Point

	{attribute 'TcIecLibraryType'}
	{attribute 'external_name' := 'F_VN_TransformCoordinatesImageToWorld_Point_GUID_EFB98558_B4AE_5C23_6CCF_F027CE21A2E4'}
	(* Transform 2D image point coordinate to 3D world coordinate (using intrinsic + extrinsic calibration results). *)
	FUNCTION F_VN_TransformCoordinatesImageToWorld_Point : HRESULT
	VAR_INPUT
		aSrcPoint	:	REFERENCE TO TcVnPoint2_LREAL;	(* Point in the image coordinate system *)
		aDestPoint	:	REFERENCE TO TcVnPoint3_LREAL;	(* Returns the point in the world coordinate system *)
		aCameraMatrix	:	REFERENCE TO TcVnMatrix3x3_LREAL;	(* 3x3 camera matrix containing the intrinsic parameters *)
		aDistortionCoefficients	:	REFERENCE TO TcVnArray8_LREAL;	(* Lens distortion coefficients [k1, k2, p1, p2, k3, k4, k5, k6] *)
		aRotationMatrix	:	REFERENCE TO TcVnMatrix3x3_LREAL;	(* 3x3 rotation matrix *)
		aTranslationVector	:	REFERENCE TO TcVnVector3_LREAL;	(* Translation vector *)
		fZ	:	LREAL;	(* z coordinate (world coordinate system) of the transformed points (0 would be at (toplevel) calibration pattern) *)
		hrPrev	:	HRESULT;	(* HRESULT indicating the result of previous operations (If SUCCEEDED(hrPrev) equals false, no operation is executed.) *)
	END_VAR

END_FUNCTION

// Functions/Geometric and Coordinate Transformations/Calibration/F_VN_TransformCoordinatesWorldToImage_Container

	{attribute 'TcIecLibraryType'}
	{attribute 'external_name' := 'F_VN_TransformCoordinatesWorldToImage_Container_GUID_AA8D71AA_9B5D_526B_6C5E_5E8EFE8E239A'}
	(* Transform 3D world coordinates to 2D image coordinates (using intrinsic + extrinsic calibration results). *)
	FUNCTION F_VN_TransformCoordinatesWorldToImage_Container : HRESULT
	VAR_INPUT
		ipSrcPoints3D	:	ITcVnContainer;	(* Container with 3D source points (TcVnPoint3_LREAL) *)
		ipDestPoints2D	:	REFERENCE TO ITcVnContainer;	(* Returns the transformed 2D points (TcVnPoint2_REAL or TcVnPoint2_DINT, depending on bInteger) *)
		aCameraMatrix	:	REFERENCE TO TcVnMatrix3x3_LREAL;	(* 3x3 camera matrix containing the intrinsic parameters *)
		aDistortionCoefficients	:	REFERENCE TO TcVnArray8_LREAL;	(* Lens distortion coefficients [k1, k2, p1, p2, k3, k4, k5, k6] *)
		aRotationMatrix	:	REFERENCE TO TcVnMatrix3x3_LREAL;	(* 3x3 rotation matrix *)
		aTranslationVector	:	REFERENCE TO TcVnVector3_LREAL;	(* Translation vector *)
		bInteger	:	BOOL;	(* Selects whether the function returns a container of TcVnPoint2_DINT or TcVnPoint2_REAL *)
		hrPrev	:	HRESULT;	(* HRESULT indicating the result of previous operations (If SUCCEEDED(hrPrev) equals false, no operation is executed.) *)
	END_VAR

END_FUNCTION

// Functions/Geometric and Coordinate Transformations/Calibration/F_VN_TransformCoordinatesWorldToImage_Point

	{attribute 'TcIecLibraryType'}
	{attribute 'external_name' := 'F_VN_TransformCoordinatesWorldToImage_Point_GUID_EEBF188A_B8B9_5909_6E01_AFD0BEADA794'}
	(* Transform 3D world coordinates to 2D image coordinates (using intrinsic + extrinsic calibration results). *)
	FUNCTION F_VN_TransformCoordinatesWorldToImage_Point : HRESULT
	VAR_INPUT
		aSrcPoint	:	REFERENCE TO TcVnPoint3_LREAL;	(* 3D source point (world coordinate system) *)
		aDestPoint	:	REFERENCE TO TcVnPoint2_REAL;	(* Returns the transformed 2D point (image coordinate system) *)
		aCameraMatrix	:	REFERENCE TO TcVnMatrix3x3_LREAL;	(* 3x3 camera matrix containing the intrinsic parameters *)
		aDistortionCoefficients	:	REFERENCE TO TcVnArray8_LREAL;	(* Lens distortion coefficients [k1, k2, p1, p2, k3, k4, k5, k6] *)
		aRotationMatrix	:	REFERENCE TO TcVnMatrix3x3_LREAL;	(* 3x3 rotation matrix *)
		aTranslationVector	:	REFERENCE TO TcVnVector3_LREAL;	(* Translation vector *)
		hrPrev	:	HRESULT;	(* HRESULT indicating the result of previous operations (If SUCCEEDED(hrPrev) equals false, no operation is executed.) *)
	END_VAR

END_FUNCTION

// Functions/Container Statistics/F_VN_MaxElementElementwise/F_VN_MaxElementElementwise_DINT

	{attribute 'TcIecLibraryType'}
	{attribute 'external_name' := 'F_VN_MaxElementElementwise_DINT_GUID_C98AF7AB_56CC_57E6_5493_B27637C0D032'}
	(* Gets the element wise maximum container element. *)
	FUNCTION F_VN_MaxElementElementwise_DINT : HRESULT
	VAR_INPUT
		ipContainer	:	ITcVnContainer;	(* Source container *)
		nMax	:	REFERENCE TO DINT;	(* Returns the requested element *)
		hrPrev	:	HRESULT;	(* HRESULT indicating the result of previous operations (If SUCCEEDED(hrPrev) equals false, no operation is executed.) *)
	END_VAR

END_FUNCTION

// Functions/Container Statistics/F_VN_MaxElementElementwise/F_VN_MaxElementElementwise_LREAL

	{attribute 'TcIecLibraryType'}
	{attribute 'external_name' := 'F_VN_MaxElementElementwise_LREAL_GUID_2A3E8EC8_F128_588A_6EE5_33C1A06A009C'}
	(* Gets the element wise maximum container element. *)
	FUNCTION F_VN_MaxElementElementwise_LREAL : HRESULT
	VAR_INPUT
		ipContainer	:	ITcVnContainer;	(* Source container *)
		fMax	:	REFERENCE TO LREAL;	(* Returns the requested element *)
		hrPrev	:	HRESULT;	(* HRESULT indicating the result of previous operations (If SUCCEEDED(hrPrev) equals false, no operation is executed.) *)
	END_VAR

END_FUNCTION

// Functions/Container Statistics/F_VN_MaxElementElementwise/F_VN_MaxElementElementwise_REAL

	{attribute 'TcIecLibraryType'}
	{attribute 'external_name' := 'F_VN_MaxElementElementwise_REAL_GUID_41CF3A3D_6549_55A9_63E5_D8722147DA12'}
	(* Gets the element wise maximum container element. *)
	FUNCTION F_VN_MaxElementElementwise_REAL : HRESULT
	VAR_INPUT
		ipContainer	:	ITcVnContainer;	(* Source container *)
		fMax	:	REFERENCE TO REAL;	(* Returns the requested element *)
		hrPrev	:	HRESULT;	(* HRESULT indicating the result of previous operations (If SUCCEEDED(hrPrev) equals false, no operation is executed.) *)
	END_VAR

END_FUNCTION

// Functions/Container Statistics/F_VN_MaxElementElementwise/F_VN_MaxElementElementwise_SINT

	{attribute 'TcIecLibraryType'}
	{attribute 'external_name' := 'F_VN_MaxElementElementwise_SINT_GUID_BF5E1168_B97B_5AA5_44C6_95FEA6EAEBE8'}
	(* Gets the element wise maximum container element. *)
	FUNCTION F_VN_MaxElementElementwise_SINT : HRESULT
	VAR_INPUT
		ipContainer	:	ITcVnContainer;	(* Source container *)
		nMax	:	REFERENCE TO SINT;	(* Returns the requested element *)
		hrPrev	:	HRESULT;	(* HRESULT indicating the result of previous operations (If SUCCEEDED(hrPrev) equals false, no operation is executed.) *)
	END_VAR

END_FUNCTION

// Functions/Container Statistics/F_VN_MaxElementElementwise/F_VN_MaxElementElementwise_TcVnPoint2_DINT

	{attribute 'TcIecLibraryType'}
	{attribute 'external_name' := 'F_VN_MaxElementElementwise_TcVnPoint2_DINT_GUID_C3B9FD32_728B_56A7_76C0_7A5C6C81DD31'}
	(* Gets the element wise maximum container element. *)
	FUNCTION F_VN_MaxElementElementwise_TcVnPoint2_DINT : HRESULT
	VAR_INPUT
		ipContainer	:	ITcVnContainer;	(* Source container *)
		aMax	:	REFERENCE TO TcVnPoint2_DINT;	(* Returns the requested element *)
		hrPrev	:	HRESULT;	(* HRESULT indicating the result of previous operations (If SUCCEEDED(hrPrev) equals false, no operation is executed.) *)
	END_VAR

END_FUNCTION

// Functions/Container Statistics/F_VN_MaxElementElementwise/F_VN_MaxElementElementwise_TcVnPoint2_LREAL

	{attribute 'TcIecLibraryType'}
	{attribute 'external_name' := 'F_VN_MaxElementElementwise_TcVnPoint2_LREAL_GUID_CDD9B01E_3E48_5636_53B6_DCE8899F5881'}
	(* Gets the element wise maximum container element. *)
	FUNCTION F_VN_MaxElementElementwise_TcVnPoint2_LREAL : HRESULT
	VAR_INPUT
		ipContainer	:	ITcVnContainer;	(* Source container *)
		aMax	:	REFERENCE TO TcVnPoint2_LREAL;	(* Returns the requested element *)
		hrPrev	:	HRESULT;	(* HRESULT indicating the result of previous operations (If SUCCEEDED(hrPrev) equals false, no operation is executed.) *)
	END_VAR

END_FUNCTION

// Functions/Container Statistics/F_VN_MaxElementElementwise/F_VN_MaxElementElementwise_TcVnPoint2_REAL

	{attribute 'TcIecLibraryType'}
	{attribute 'external_name' := 'F_VN_MaxElementElementwise_TcVnPoint2_REAL_GUID_6620B218_E936_5552_713C_BF3A14021415'}
	(* Gets the element wise maximum container element. *)
	FUNCTION F_VN_MaxElementElementwise_TcVnPoint2_REAL : HRESULT
	VAR_INPUT
		ipContainer	:	ITcVnContainer;	(* Source container *)
		aMax	:	REFERENCE TO TcVnPoint2_REAL;	(* Returns the requested element *)
		hrPrev	:	HRESULT;	(* HRESULT indicating the result of previous operations (If SUCCEEDED(hrPrev) equals false, no operation is executed.) *)
	END_VAR

END_FUNCTION

// Functions/Container Statistics/F_VN_MaxElementElementwise/F_VN_MaxElementElementwise_TcVnPoint3_LREAL

	{attribute 'TcIecLibraryType'}
	{attribute 'external_name' := 'F_VN_MaxElementElementwise_TcVnPoint3_LREAL_GUID_6275D7C0_5FF9_5B4F_527C_4C477599B2B3'}
	(* Gets the element wise maximum container element. *)
	FUNCTION F_VN_MaxElementElementwise_TcVnPoint3_LREAL : HRESULT
	VAR_INPUT
		ipContainer	:	ITcVnContainer;	(* Source container *)
		aMax	:	REFERENCE TO TcVnPoint3_LREAL;	(* Returns the requested element *)
		hrPrev	:	HRESULT;	(* HRESULT indicating the result of previous operations (If SUCCEEDED(hrPrev) equals false, no operation is executed.) *)
	END_VAR

END_FUNCTION

// Functions/Container Statistics/F_VN_MaxElementElementwise/F_VN_MaxElementElementwise_TcVnPoint3_REAL

	{attribute 'TcIecLibraryType'}
	{attribute 'external_name' := 'F_VN_MaxElementElementwise_TcVnPoint3_REAL_GUID_95A8C032_C8FF_5AE3_5557_6C399C5D237E'}
	(* Gets the element wise maximum container element. *)
	FUNCTION F_VN_MaxElementElementwise_TcVnPoint3_REAL : HRESULT
	VAR_INPUT
		ipContainer	:	ITcVnContainer;	(* Source container *)
		aMax	:	REFERENCE TO TcVnPoint3_REAL;	(* Returns the requested element *)
		hrPrev	:	HRESULT;	(* HRESULT indicating the result of previous operations (If SUCCEEDED(hrPrev) equals false, no operation is executed.) *)
	END_VAR

END_FUNCTION

// Functions/Container Statistics/F_VN_MaxElementElementwise/F_VN_MaxElementElementwise_TcVnVector2_DINT

	{attribute 'TcIecLibraryType'}
	{attribute 'external_name' := 'F_VN_MaxElementElementwise_TcVnVector2_DINT_GUID_ABD64B03_A5A7_5CA8_45E0_955D0270CCFB'}
	(* Gets the element wise maximum container element. *)
	FUNCTION F_VN_MaxElementElementwise_TcVnVector2_DINT : HRESULT
	VAR_INPUT
		ipContainer	:	ITcVnContainer;	(* Source container *)
		aMax	:	REFERENCE TO TcVnVector2_DINT;	(* Returns the requested element *)
		hrPrev	:	HRESULT;	(* HRESULT indicating the result of previous operations (If SUCCEEDED(hrPrev) equals false, no operation is executed.) *)
	END_VAR

END_FUNCTION

// Functions/Container Statistics/F_VN_MaxElementElementwise/F_VN_MaxElementElementwise_TcVnVector2_REAL

	{attribute 'TcIecLibraryType'}
	{attribute 'external_name' := 'F_VN_MaxElementElementwise_TcVnVector2_REAL_GUID_C54A6415_4011_506E_4571_CC593C6D6900'}
	(* Gets the element wise maximum container element. *)
	FUNCTION F_VN_MaxElementElementwise_TcVnVector2_REAL : HRESULT
	VAR_INPUT
		ipContainer	:	ITcVnContainer;	(* Source container *)
		aMax	:	REFERENCE TO TcVnVector2_REAL;	(* Returns the requested element *)
		hrPrev	:	HRESULT;	(* HRESULT indicating the result of previous operations (If SUCCEEDED(hrPrev) equals false, no operation is executed.) *)
	END_VAR

END_FUNCTION

// Functions/Container Statistics/F_VN_MaxElementElementwise/F_VN_MaxElementElementwise_TcVnVector3_REAL

	{attribute 'TcIecLibraryType'}
	{attribute 'external_name' := 'F_VN_MaxElementElementwise_TcVnVector3_REAL_GUID_F202B0FF_602F_510A_769F_B41F07A62490'}
	(* Gets the element wise maximum container element. *)
	FUNCTION F_VN_MaxElementElementwise_TcVnVector3_REAL : HRESULT
	VAR_INPUT
		ipContainer	:	ITcVnContainer;	(* Source container *)
		aMax	:	REFERENCE TO TcVnVector3_REAL;	(* Returns the requested element *)
		hrPrev	:	HRESULT;	(* HRESULT indicating the result of previous operations (If SUCCEEDED(hrPrev) equals false, no operation is executed.) *)
	END_VAR

END_FUNCTION

// Functions/Container Statistics/F_VN_MaxElementElementwise/F_VN_MaxElementElementwise_TcVnVector4_DINT

	{attribute 'TcIecLibraryType'}
	{attribute 'external_name' := 'F_VN_MaxElementElementwise_TcVnVector4_DINT_GUID_3E877F0E_EE63_58D2_588F_14A056CA63DF'}
	(* Gets the element wise maximum container element. *)
	FUNCTION F_VN_MaxElementElementwise_TcVnVector4_DINT : HRESULT
	VAR_INPUT
		ipContainer	:	ITcVnContainer;	(* Source container *)
		aMax	:	REFERENCE TO TcVnVector4_DINT;	(* Returns the requested element *)
		hrPrev	:	HRESULT;	(* HRESULT indicating the result of previous operations (If SUCCEEDED(hrPrev) equals false, no operation is executed.) *)
	END_VAR

END_FUNCTION

// Functions/Container Statistics/F_VN_MaxElementElementwise/F_VN_MaxElementElementwise_TcVnVector4_LREAL

	{attribute 'TcIecLibraryType'}
	{attribute 'external_name' := 'F_VN_MaxElementElementwise_TcVnVector4_LREAL_GUID_04B38A17_398B_57CD_6E54_A70CF9ED1BC4'}
	(* Gets the element wise maximum container element. *)
	FUNCTION F_VN_MaxElementElementwise_TcVnVector4_LREAL : HRESULT
	VAR_INPUT
		ipContainer	:	ITcVnContainer;	(* Source container *)
		aMax	:	REFERENCE TO TcVnVector4_LREAL;	(* Returns the requested element *)
		hrPrev	:	HRESULT;	(* HRESULT indicating the result of previous operations (If SUCCEEDED(hrPrev) equals false, no operation is executed.) *)
	END_VAR

END_FUNCTION

// Functions/Container Statistics/F_VN_MaxElementElementwise/F_VN_MaxElementElementwise_UDINT

	{attribute 'TcIecLibraryType'}
	{attribute 'external_name' := 'F_VN_MaxElementElementwise_UDINT_GUID_DCFE7FDD_7E28_5318_75DD_AEF10212B0F2'}
	(* Gets the element wise maximum container element. *)
	FUNCTION F_VN_MaxElementElementwise_UDINT : HRESULT
	VAR_INPUT
		ipContainer	:	ITcVnContainer;	(* Source container *)
		nMax	:	REFERENCE TO UDINT;	(* Returns the requested element *)
		hrPrev	:	HRESULT;	(* HRESULT indicating the result of previous operations (If SUCCEEDED(hrPrev) equals false, no operation is executed.) *)
	END_VAR

END_FUNCTION

// Functions/Container Statistics/F_VN_MaxElementElementwise/F_VN_MaxElementElementwise_ULINT

	{attribute 'TcIecLibraryType'}
	{attribute 'external_name' := 'F_VN_MaxElementElementwise_ULINT_GUID_8AE2A4D1_D193_57D6_7F8A_F7EA65B0A184'}
	(* Gets the element wise maximum container element. *)
	FUNCTION F_VN_MaxElementElementwise_ULINT : HRESULT
	VAR_INPUT
		ipContainer	:	ITcVnContainer;	(* Source container *)
		nMax	:	REFERENCE TO ULINT;	(* Returns the requested element *)
		hrPrev	:	HRESULT;	(* HRESULT indicating the result of previous operations (If SUCCEEDED(hrPrev) equals false, no operation is executed.) *)
	END_VAR

END_FUNCTION

// Functions/Container Statistics/F_VN_MedianElementElementwise/F_VN_MedianElementElementwise_DINT

	{attribute 'TcIecLibraryType'}
	{attribute 'external_name' := 'F_VN_MedianElementElementwise_DINT_GUID_DA1F72DD_588C_51B7_64E9_8978E44BD5F1'}
	(* Gets the element wise median container element. *)
	FUNCTION F_VN_MedianElementElementwise_DINT : HRESULT
	VAR_INPUT
		ipContainer	:	ITcVnContainer;	(* Source container *)
		nMedian	:	REFERENCE TO DINT;	(* Returns the requested element *)
		hrPrev	:	HRESULT;	(* HRESULT indicating the result of previous operations (If SUCCEEDED(hrPrev) equals false, no operation is executed.) *)
	END_VAR

END_FUNCTION

// Functions/Container Statistics/F_VN_MedianElementElementwise/F_VN_MedianElementElementwise_LREAL

	{attribute 'TcIecLibraryType'}
	{attribute 'external_name' := 'F_VN_MedianElementElementwise_LREAL_GUID_46D4EAFE_2724_5A02_4781_42A7C3D5D80D'}
	(* Gets the element wise median container element. *)
	FUNCTION F_VN_MedianElementElementwise_LREAL : HRESULT
	VAR_INPUT
		ipContainer	:	ITcVnContainer;	(* Source container *)
		fMedian	:	REFERENCE TO LREAL;	(* Returns the requested element *)
		hrPrev	:	HRESULT;	(* HRESULT indicating the result of previous operations (If SUCCEEDED(hrPrev) equals false, no operation is executed.) *)
	END_VAR

END_FUNCTION

// Functions/Container Statistics/F_VN_MedianElementElementwise/F_VN_MedianElementElementwise_REAL

	{attribute 'TcIecLibraryType'}
	{attribute 'external_name' := 'F_VN_MedianElementElementwise_REAL_GUID_D26B0D46_2325_5A74_60AD_D47FF9473345'}
	(* Gets the element wise median container element. *)
	FUNCTION F_VN_MedianElementElementwise_REAL : HRESULT
	VAR_INPUT
		ipContainer	:	ITcVnContainer;	(* Source container *)
		fMedian	:	REFERENCE TO REAL;	(* Returns the requested element *)
		hrPrev	:	HRESULT;	(* HRESULT indicating the result of previous operations (If SUCCEEDED(hrPrev) equals false, no operation is executed.) *)
	END_VAR

END_FUNCTION

// Functions/Container Statistics/F_VN_MedianElementElementwise/F_VN_MedianElementElementwise_SINT

	{attribute 'TcIecLibraryType'}
	{attribute 'external_name' := 'F_VN_MedianElementElementwise_SINT_GUID_54DEAA27_B966_5EF6_4D61_204F007FC7AB'}
	(* Gets the element wise median container element. *)
	FUNCTION F_VN_MedianElementElementwise_SINT : HRESULT
	VAR_INPUT
		ipContainer	:	ITcVnContainer;	(* Source container *)
		nMedian	:	REFERENCE TO SINT;	(* Returns the requested element *)
		hrPrev	:	HRESULT;	(* HRESULT indicating the result of previous operations (If SUCCEEDED(hrPrev) equals false, no operation is executed.) *)
	END_VAR

END_FUNCTION

// Functions/Container Statistics/F_VN_MedianElementElementwise/F_VN_MedianElementElementwise_TcVnPoint2_DINT

	{attribute 'TcIecLibraryType'}
	{attribute 'external_name' := 'F_VN_MedianElementElementwise_TcVnPoint2_DINT_GUID_50ECD82C_F9AB_513D_6881_3047368548C6'}
	(* Gets the element wise median container element. *)
	FUNCTION F_VN_MedianElementElementwise_TcVnPoint2_DINT : HRESULT
	VAR_INPUT
		ipContainer	:	ITcVnContainer;	(* Source container *)
		aMedian	:	REFERENCE TO TcVnPoint2_DINT;	(* Returns the requested element *)
		hrPrev	:	HRESULT;	(* HRESULT indicating the result of previous operations (If SUCCEEDED(hrPrev) equals false, no operation is executed.) *)
	END_VAR

END_FUNCTION

// Functions/Container Statistics/F_VN_MedianElementElementwise/F_VN_MedianElementElementwise_TcVnPoint2_LREAL

	{attribute 'TcIecLibraryType'}
	{attribute 'external_name' := 'F_VN_MedianElementElementwise_TcVnPoint2_LREAL_GUID_AB1F33BA_E700_56B8_7125_B5A8930EC214'}
	(* Gets the element wise median container element. *)
	FUNCTION F_VN_MedianElementElementwise_TcVnPoint2_LREAL : HRESULT
	VAR_INPUT
		ipContainer	:	ITcVnContainer;	(* Source container *)
		aMedian	:	REFERENCE TO TcVnPoint2_LREAL;	(* Returns the requested element *)
		hrPrev	:	HRESULT;	(* HRESULT indicating the result of previous operations (If SUCCEEDED(hrPrev) equals false, no operation is executed.) *)
	END_VAR

END_FUNCTION

// Functions/Container Statistics/F_VN_MedianElementElementwise/F_VN_MedianElementElementwise_TcVnPoint2_REAL

	{attribute 'TcIecLibraryType'}
	{attribute 'external_name' := 'F_VN_MedianElementElementwise_TcVnPoint2_REAL_GUID_0BE687E7_949D_5F6D_4211_FC3657AC0314'}
	(* Gets the element wise median container element. *)
	FUNCTION F_VN_MedianElementElementwise_TcVnPoint2_REAL : HRESULT
	VAR_INPUT
		ipContainer	:	ITcVnContainer;	(* Source container *)
		aMedian	:	REFERENCE TO TcVnPoint2_REAL;	(* Returns the requested element *)
		hrPrev	:	HRESULT;	(* HRESULT indicating the result of previous operations (If SUCCEEDED(hrPrev) equals false, no operation is executed.) *)
	END_VAR

END_FUNCTION

// Functions/Container Statistics/F_VN_MedianElementElementwise/F_VN_MedianElementElementwise_TcVnPoint3_LREAL

	{attribute 'TcIecLibraryType'}
	{attribute 'external_name' := 'F_VN_MedianElementElementwise_TcVnPoint3_LREAL_GUID_02FFC7EE_9FAB_51D6_77C7_C022E7CD019F'}
	(* Gets the element wise median container element. *)
	FUNCTION F_VN_MedianElementElementwise_TcVnPoint3_LREAL : HRESULT
	VAR_INPUT
		ipContainer	:	ITcVnContainer;	(* Source container *)
		aMedian	:	REFERENCE TO TcVnPoint3_LREAL;	(* Returns the requested element *)
		hrPrev	:	HRESULT;	(* HRESULT indicating the result of previous operations (If SUCCEEDED(hrPrev) equals false, no operation is executed.) *)
	END_VAR

END_FUNCTION

// Functions/Container Statistics/F_VN_MedianElementElementwise/F_VN_MedianElementElementwise_TcVnPoint3_REAL

	{attribute 'TcIecLibraryType'}
	{attribute 'external_name' := 'F_VN_MedianElementElementwise_TcVnPoint3_REAL_GUID_86DADCA8_CA21_5245_7859_54BF274A636C'}
	(* Gets the element wise median container element. *)
	FUNCTION F_VN_MedianElementElementwise_TcVnPoint3_REAL : HRESULT
	VAR_INPUT
		ipContainer	:	ITcVnContainer;	(* Source container *)
		aMedian	:	REFERENCE TO TcVnPoint3_REAL;	(* Returns the requested element *)
		hrPrev	:	HRESULT;	(* HRESULT indicating the result of previous operations (If SUCCEEDED(hrPrev) equals false, no operation is executed.) *)
	END_VAR

END_FUNCTION

// Functions/Container Statistics/F_VN_MedianElementElementwise/F_VN_MedianElementElementwise_TcVnVector2_DINT

	{attribute 'TcIecLibraryType'}
	{attribute 'external_name' := 'F_VN_MedianElementElementwise_TcVnVector2_DINT_GUID_7DF2C177_1A12_561F_45DD_B9FC856B207C'}
	(* Gets the element wise median container element. *)
	FUNCTION F_VN_MedianElementElementwise_TcVnVector2_DINT : HRESULT
	VAR_INPUT
		ipContainer	:	ITcVnContainer;	(* Source container *)
		aMedian	:	REFERENCE TO TcVnVector2_DINT;	(* Returns the requested element *)
		hrPrev	:	HRESULT;	(* HRESULT indicating the result of previous operations (If SUCCEEDED(hrPrev) equals false, no operation is executed.) *)
	END_VAR

END_FUNCTION

// Functions/Container Statistics/F_VN_MedianElementElementwise/F_VN_MedianElementElementwise_TcVnVector2_REAL

	{attribute 'TcIecLibraryType'}
	{attribute 'external_name' := 'F_VN_MedianElementElementwise_TcVnVector2_REAL_GUID_755C4BCF_5E27_5E93_4D95_7A57E08FC6DE'}
	(* Gets the element wise median container element. *)
	FUNCTION F_VN_MedianElementElementwise_TcVnVector2_REAL : HRESULT
	VAR_INPUT
		ipContainer	:	ITcVnContainer;	(* Source container *)
		aMedian	:	REFERENCE TO TcVnVector2_REAL;	(* Returns the requested element *)
		hrPrev	:	HRESULT;	(* HRESULT indicating the result of previous operations (If SUCCEEDED(hrPrev) equals false, no operation is executed.) *)
	END_VAR

END_FUNCTION

// Functions/Container Statistics/F_VN_MedianElementElementwise/F_VN_MedianElementElementwise_TcVnVector3_REAL

	{attribute 'TcIecLibraryType'}
	{attribute 'external_name' := 'F_VN_MedianElementElementwise_TcVnVector3_REAL_GUID_BD2CB986_6469_57E2_48A9_3DF0A316F731'}
	(* Gets the element wise median container element. *)
	FUNCTION F_VN_MedianElementElementwise_TcVnVector3_REAL : HRESULT
	VAR_INPUT
		ipContainer	:	ITcVnContainer;	(* Source container *)
		aMedian	:	REFERENCE TO TcVnVector3_REAL;	(* Returns the requested element *)
		hrPrev	:	HRESULT;	(* HRESULT indicating the result of previous operations (If SUCCEEDED(hrPrev) equals false, no operation is executed.) *)
	END_VAR

END_FUNCTION

// Functions/Container Statistics/F_VN_MedianElementElementwise/F_VN_MedianElementElementwise_TcVnVector4_DINT

	{attribute 'TcIecLibraryType'}
	{attribute 'external_name' := 'F_VN_MedianElementElementwise_TcVnVector4_DINT_GUID_9C185F4B_BCB7_5CEC_4B8B_5D1C16F3CF0D'}
	(* Gets the element wise median container element. *)
	FUNCTION F_VN_MedianElementElementwise_TcVnVector4_DINT : HRESULT
	VAR_INPUT
		ipContainer	:	ITcVnContainer;	(* Source container *)
		aMedian	:	REFERENCE TO TcVnVector4_DINT;	(* Returns the requested element *)
		hrPrev	:	HRESULT;	(* HRESULT indicating the result of previous operations (If SUCCEEDED(hrPrev) equals false, no operation is executed.) *)
	END_VAR

END_FUNCTION

// Functions/Container Statistics/F_VN_MedianElementElementwise/F_VN_MedianElementElementwise_TcVnVector4_LREAL

	{attribute 'TcIecLibraryType'}
	{attribute 'external_name' := 'F_VN_MedianElementElementwise_TcVnVector4_LREAL_GUID_91D3F6A5_E7D4_5763_7491_D28EB3F120F0'}
	(* Gets the element wise median container element. *)
	FUNCTION F_VN_MedianElementElementwise_TcVnVector4_LREAL : HRESULT
	VAR_INPUT
		ipContainer	:	ITcVnContainer;	(* Source container *)
		aMedian	:	REFERENCE TO TcVnVector4_LREAL;	(* Returns the requested element *)
		hrPrev	:	HRESULT;	(* HRESULT indicating the result of previous operations (If SUCCEEDED(hrPrev) equals false, no operation is executed.) *)
	END_VAR

END_FUNCTION

// Functions/Container Statistics/F_VN_MedianElementElementwise/F_VN_MedianElementElementwise_UDINT

	{attribute 'TcIecLibraryType'}
	{attribute 'external_name' := 'F_VN_MedianElementElementwise_UDINT_GUID_68724BC0_8CFB_5EF5_4CEA_15856B15F8B0'}
	(* Gets the element wise median container element. *)
	FUNCTION F_VN_MedianElementElementwise_UDINT : HRESULT
	VAR_INPUT
		ipContainer	:	ITcVnContainer;	(* Source container *)
		nMedian	:	REFERENCE TO UDINT;	(* Returns the requested element *)
		hrPrev	:	HRESULT;	(* HRESULT indicating the result of previous operations (If SUCCEEDED(hrPrev) equals false, no operation is executed.) *)
	END_VAR

END_FUNCTION

// Functions/Container Statistics/F_VN_MedianElementElementwise/F_VN_MedianElementElementwise_ULINT

	{attribute 'TcIecLibraryType'}
	{attribute 'external_name' := 'F_VN_MedianElementElementwise_ULINT_GUID_7D7A4BF7_B39D_530D_741D_D7364D68B1D0'}
	(* Gets the element wise median container element. *)
	FUNCTION F_VN_MedianElementElementwise_ULINT : HRESULT
	VAR_INPUT
		ipContainer	:	ITcVnContainer;	(* Source container *)
		nMedian	:	REFERENCE TO ULINT;	(* Returns the requested element *)
		hrPrev	:	HRESULT;	(* HRESULT indicating the result of previous operations (If SUCCEEDED(hrPrev) equals false, no operation is executed.) *)
	END_VAR

END_FUNCTION

// Functions/Container Statistics/F_VN_MinElementElementwise/F_VN_MinElementElementwise_DINT

	{attribute 'TcIecLibraryType'}
	{attribute 'external_name' := 'F_VN_MinElementElementwise_DINT_GUID_8DE38545_260F_5AD9_5C53_19D483529A10'}
	(* Gets the element wise minimum container element. *)
	FUNCTION F_VN_MinElementElementwise_DINT : HRESULT
	VAR_INPUT
		ipContainer	:	ITcVnContainer;	(* Source container *)
		nMin	:	REFERENCE TO DINT;	(* Returns the requested element *)
		hrPrev	:	HRESULT;	(* HRESULT indicating the result of previous operations (If SUCCEEDED(hrPrev) equals false, no operation is executed.) *)
	END_VAR

END_FUNCTION

// Functions/Container Statistics/F_VN_MinElementElementwise/F_VN_MinElementElementwise_LREAL

	{attribute 'TcIecLibraryType'}
	{attribute 'external_name' := 'F_VN_MinElementElementwise_LREAL_GUID_32607C5D_7D5B_5DDA_540E_F578A49B9CBE'}
	(* Gets the element wise minimum container element. *)
	FUNCTION F_VN_MinElementElementwise_LREAL : HRESULT
	VAR_INPUT
		ipContainer	:	ITcVnContainer;	(* Source container *)
		fMin	:	REFERENCE TO LREAL;	(* Returns the requested element *)
		hrPrev	:	HRESULT;	(* HRESULT indicating the result of previous operations (If SUCCEEDED(hrPrev) equals false, no operation is executed.) *)
	END_VAR

END_FUNCTION

// Functions/Container Statistics/F_VN_MinElementElementwise/F_VN_MinElementElementwise_REAL

	{attribute 'TcIecLibraryType'}
	{attribute 'external_name' := 'F_VN_MinElementElementwise_REAL_GUID_B6B3F1FC_0026_524B_61AB_C192437E32B2'}
	(* Gets the element wise minimum container element. *)
	FUNCTION F_VN_MinElementElementwise_REAL : HRESULT
	VAR_INPUT
		ipContainer	:	ITcVnContainer;	(* Source container *)
		fMin	:	REFERENCE TO REAL;	(* Returns the requested element *)
		hrPrev	:	HRESULT;	(* HRESULT indicating the result of previous operations (If SUCCEEDED(hrPrev) equals false, no operation is executed.) *)
	END_VAR

END_FUNCTION

// Functions/Container Statistics/F_VN_MinElementElementwise/F_VN_MinElementElementwise_SINT

	{attribute 'TcIecLibraryType'}
	{attribute 'external_name' := 'F_VN_MinElementElementwise_SINT_GUID_DDB85631_4837_5612_5A7F_4904CD7BF315'}
	(* Gets the element wise minimum container element. *)
	FUNCTION F_VN_MinElementElementwise_SINT : HRESULT
	VAR_INPUT
		ipContainer	:	ITcVnContainer;	(* Source container *)
		nMin	:	REFERENCE TO SINT;	(* Returns the requested element *)
		hrPrev	:	HRESULT;	(* HRESULT indicating the result of previous operations (If SUCCEEDED(hrPrev) equals false, no operation is executed.) *)
	END_VAR

END_FUNCTION

// Functions/Container Statistics/F_VN_MinElementElementwise/F_VN_MinElementElementwise_TcVnPoint2_DINT

	{attribute 'TcIecLibraryType'}
	{attribute 'external_name' := 'F_VN_MinElementElementwise_TcVnPoint2_DINT_GUID_FD7CBA6F_B087_5788_5D3E_B8E8B415110F'}
	(* Gets the element wise minimum container element. *)
	FUNCTION F_VN_MinElementElementwise_TcVnPoint2_DINT : HRESULT
	VAR_INPUT
		ipContainer	:	ITcVnContainer;	(* Source container *)
		aMin	:	REFERENCE TO TcVnPoint2_DINT;	(* Returns the requested element *)
		hrPrev	:	HRESULT;	(* HRESULT indicating the result of previous operations (If SUCCEEDED(hrPrev) equals false, no operation is executed.) *)
	END_VAR

END_FUNCTION

// Functions/Container Statistics/F_VN_MinElementElementwise/F_VN_MinElementElementwise_TcVnPoint2_LREAL

	{attribute 'TcIecLibraryType'}
	{attribute 'external_name' := 'F_VN_MinElementElementwise_TcVnPoint2_LREAL_GUID_694998C8_F596_512F_63D7_A7F0D78E30CF'}
	(* Gets the element wise minimum container element. *)
	FUNCTION F_VN_MinElementElementwise_TcVnPoint2_LREAL : HRESULT
	VAR_INPUT
		ipContainer	:	ITcVnContainer;	(* Source container *)
		aMin	:	REFERENCE TO TcVnPoint2_LREAL;	(* Returns the requested element *)
		hrPrev	:	HRESULT;	(* HRESULT indicating the result of previous operations (If SUCCEEDED(hrPrev) equals false, no operation is executed.) *)
	END_VAR

END_FUNCTION

// Functions/Container Statistics/F_VN_MinElementElementwise/F_VN_MinElementElementwise_TcVnPoint2_REAL

	{attribute 'TcIecLibraryType'}
	{attribute 'external_name' := 'F_VN_MinElementElementwise_TcVnPoint2_REAL_GUID_89734DDD_AB44_5650_4DC9_DED1CADE5F6A'}
	(* Gets the element wise minimum container element. *)
	FUNCTION F_VN_MinElementElementwise_TcVnPoint2_REAL : HRESULT
	VAR_INPUT
		ipContainer	:	ITcVnContainer;	(* Source container *)
		aMin	:	REFERENCE TO TcVnPoint2_REAL;	(* Returns the requested element *)
		hrPrev	:	HRESULT;	(* HRESULT indicating the result of previous operations (If SUCCEEDED(hrPrev) equals false, no operation is executed.) *)
	END_VAR

END_FUNCTION

// Functions/Container Statistics/F_VN_MinElementElementwise/F_VN_MinElementElementwise_TcVnPoint3_LREAL

	{attribute 'TcIecLibraryType'}
	{attribute 'external_name' := 'F_VN_MinElementElementwise_TcVnPoint3_LREAL_GUID_439E37E3_1D61_5E38_5470_F03EF78C86A0'}
	(* Gets the element wise minimum container element. *)
	FUNCTION F_VN_MinElementElementwise_TcVnPoint3_LREAL : HRESULT
	VAR_INPUT
		ipContainer	:	ITcVnContainer;	(* Source container *)
		aMin	:	REFERENCE TO TcVnPoint3_LREAL;	(* Returns the requested element *)
		hrPrev	:	HRESULT;	(* HRESULT indicating the result of previous operations (If SUCCEEDED(hrPrev) equals false, no operation is executed.) *)
	END_VAR

END_FUNCTION

// Functions/Container Statistics/F_VN_MinElementElementwise/F_VN_MinElementElementwise_TcVnPoint3_REAL

	{attribute 'TcIecLibraryType'}
	{attribute 'external_name' := 'F_VN_MinElementElementwise_TcVnPoint3_REAL_GUID_E5DB769A_4608_50F8_6435_647744A5DC4F'}
	(* Gets the element wise minimum container element. *)
	FUNCTION F_VN_MinElementElementwise_TcVnPoint3_REAL : HRESULT
	VAR_INPUT
		ipContainer	:	ITcVnContainer;	(* Source container *)
		aMin	:	REFERENCE TO TcVnPoint3_REAL;	(* Returns the requested element *)
		hrPrev	:	HRESULT;	(* HRESULT indicating the result of previous operations (If SUCCEEDED(hrPrev) equals false, no operation is executed.) *)
	END_VAR

END_FUNCTION

// Functions/Container Statistics/F_VN_MinElementElementwise/F_VN_MinElementElementwise_TcVnVector2_DINT

	{attribute 'TcIecLibraryType'}
	{attribute 'external_name' := 'F_VN_MinElementElementwise_TcVnVector2_DINT_GUID_B945DF5C_DF9C_5DF1_47E7_7725761203B6'}
	(* Gets the element wise minimum container element. *)
	FUNCTION F_VN_MinElementElementwise_TcVnVector2_DINT : HRESULT
	VAR_INPUT
		ipContainer	:	ITcVnContainer;	(* Source container *)
		aMin	:	REFERENCE TO TcVnVector2_DINT;	(* Returns the requested element *)
		hrPrev	:	HRESULT;	(* HRESULT indicating the result of previous operations (If SUCCEEDED(hrPrev) equals false, no operation is executed.) *)
	END_VAR

END_FUNCTION

// Functions/Container Statistics/F_VN_MinElementElementwise/F_VN_MinElementElementwise_TcVnVector2_REAL

	{attribute 'TcIecLibraryType'}
	{attribute 'external_name' := 'F_VN_MinElementElementwise_TcVnVector2_REAL_GUID_76999C3D_368D_576E_5E6B_9FFF8CFBBC6C'}
	(* Gets the element wise minimum container element. *)
	FUNCTION F_VN_MinElementElementwise_TcVnVector2_REAL : HRESULT
	VAR_INPUT
		ipContainer	:	ITcVnContainer;	(* Source container *)
		aMin	:	REFERENCE TO TcVnVector2_REAL;	(* Returns the requested element *)
		hrPrev	:	HRESULT;	(* HRESULT indicating the result of previous operations (If SUCCEEDED(hrPrev) equals false, no operation is executed.) *)
	END_VAR

END_FUNCTION

// Functions/Container Statistics/F_VN_MinElementElementwise/F_VN_MinElementElementwise_TcVnVector3_REAL

	{attribute 'TcIecLibraryType'}
	{attribute 'external_name' := 'F_VN_MinElementElementwise_TcVnVector3_REAL_GUID_3F494C79_A1E6_532C_4282_4C1BC3C80519'}
	(* Gets the element wise minimum container element. *)
	FUNCTION F_VN_MinElementElementwise_TcVnVector3_REAL : HRESULT
	VAR_INPUT
		ipContainer	:	ITcVnContainer;	(* Source container *)
		aMin	:	REFERENCE TO TcVnVector3_REAL;	(* Returns the requested element *)
		hrPrev	:	HRESULT;	(* HRESULT indicating the result of previous operations (If SUCCEEDED(hrPrev) equals false, no operation is executed.) *)
	END_VAR

END_FUNCTION

// Functions/Container Statistics/F_VN_MinElementElementwise/F_VN_MinElementElementwise_TcVnVector4_DINT

	{attribute 'TcIecLibraryType'}
	{attribute 'external_name' := 'F_VN_MinElementElementwise_TcVnVector4_DINT_GUID_B9FACC92_D778_5505_4FCB_C7289860BC2B'}
	(* Gets the element wise minimum container element. *)
	FUNCTION F_VN_MinElementElementwise_TcVnVector4_DINT : HRESULT
	VAR_INPUT
		ipContainer	:	ITcVnContainer;	(* Source container *)
		aMin	:	REFERENCE TO TcVnVector4_DINT;	(* Returns the requested element *)
		hrPrev	:	HRESULT;	(* HRESULT indicating the result of previous operations (If SUCCEEDED(hrPrev) equals false, no operation is executed.) *)
	END_VAR

END_FUNCTION

// Functions/Container Statistics/F_VN_MinElementElementwise/F_VN_MinElementElementwise_TcVnVector4_LREAL

	{attribute 'TcIecLibraryType'}
	{attribute 'external_name' := 'F_VN_MinElementElementwise_TcVnVector4_LREAL_GUID_3F31C1C1_D20E_52CB_643E_B3F82117107C'}
	(* Gets the element wise minimum container element. *)
	FUNCTION F_VN_MinElementElementwise_TcVnVector4_LREAL : HRESULT
	VAR_INPUT
		ipContainer	:	ITcVnContainer;	(* Source container *)
		aMin	:	REFERENCE TO TcVnVector4_LREAL;	(* Returns the requested element *)
		hrPrev	:	HRESULT;	(* HRESULT indicating the result of previous operations (If SUCCEEDED(hrPrev) equals false, no operation is executed.) *)
	END_VAR

END_FUNCTION

// Functions/Container Statistics/F_VN_MinElementElementwise/F_VN_MinElementElementwise_UDINT

	{attribute 'TcIecLibraryType'}
	{attribute 'external_name' := 'F_VN_MinElementElementwise_UDINT_GUID_8363C8DF_E485_527A_67C0_33BBE74C38A0'}
	(* Gets the element wise minimum container element. *)
	FUNCTION F_VN_MinElementElementwise_UDINT : HRESULT
	VAR_INPUT
		ipContainer	:	ITcVnContainer;	(* Source container *)
		nMin	:	REFERENCE TO UDINT;	(* Returns the requested element *)
		hrPrev	:	HRESULT;	(* HRESULT indicating the result of previous operations (If SUCCEEDED(hrPrev) equals false, no operation is executed.) *)
	END_VAR

END_FUNCTION

// Functions/Container Statistics/F_VN_MinElementElementwise/F_VN_MinElementElementwise_ULINT

	{attribute 'TcIecLibraryType'}
	{attribute 'external_name' := 'F_VN_MinElementElementwise_ULINT_GUID_138AB482_D2C4_5CC8_6F04_CBCABE8D6EF1'}
	(* Gets the element wise minimum container element. *)
	FUNCTION F_VN_MinElementElementwise_ULINT : HRESULT
	VAR_INPUT
		ipContainer	:	ITcVnContainer;	(* Source container *)
		nMin	:	REFERENCE TO ULINT;	(* Returns the requested element *)
		hrPrev	:	HRESULT;	(* HRESULT indicating the result of previous operations (If SUCCEEDED(hrPrev) equals false, no operation is executed.) *)
	END_VAR

END_FUNCTION
